# B&R Automation Studio project RS15_RX_30005_r00
Automation Studio 3.0.90.22 SP04; D.M. Le 24/08/2012 RS15_RX30005
Current program in the machine. End of commissioning. 
Customer IP config set

## Configuration Config1

CPU 5PPC2200.AL14-000, AutomationRuntime H4.91, Build 6.3.0, Safety 0.0, Vc V4.73.2

### Task classes (Cpu.sw)
```
Cyclic#1 (cycle 6000 us, tolerance 6000 us):
  GlobProgCa <- BagMachine_Section.GlobProgCalc.prg
  Alarms1 <- SupervisoryControl_Section.Alarm_Section.Alarms1.prg
  MainAlarms <- SupervisoryControl_Section.Alarm_Section.MainAlarms.prg
  Perf_Gen <- BagMachine_Section.Perf.Perf_Gen.prg
  A0_Basic <- BagMachine_Section.Servo_Power_Supply.Axis0.A0_Basic.prg
  A1_Basic <- BagMachine_Section.Perf.Axis1.A1_Basic.prg
  A2_Basic <- BagMachine_Section.FP.Axis2.A2_Basic.prg
  A3_Basic <- BagMachine_Section.Holding.Axis3.A3_Basic.prg
  A4_Basic <- BagMachine_Section.Tearing.Axis4.A4_Basic.prg
  A5_Basic <- BagMachine_Section.EntryPull.Axis5.A5_Basic.prg
  A5_Reg1 <- BagMachine_Section.EntryPull.Registration.A5_Reg1.prg
  A6_Basic <- BagMachine_Section.ExitPull.Axis6.A6_Basic.prg
  A7_Basic <- BagMachine_Section.Drum.Axis7.A7_Basic.prg
  A8_Basic <- BagMachine_Section.ColdMicroPerf.Axis8.A8_Basic.prg [disabled]
  A9_Basic <- BagMachine_Section.MasterAxis.A9_Init.A9_Basic.prg
  A11_Basic <- BagMachine_Section.Perf.Axis11_VirtualAxis.A11_Basic.prg
  A12_Basic <- BagMachine_Section.EnvBag.Axis12.A12_Basic.prg [disabled]
  A13_Basic <- BagMachine_Section.EnvBag.Axis13.A13_Basic.prg [disabled]
  A15_Basic <- BagMachine_Section.HotMicroPerf.Axis15.A15_Basic.prg [disabled]
  A1_Automat <- BagMachine_Section.Perf.Axis1.A1_Automat.prg
  A1_Automa1 <- BagMachine_Section.Perf.Axis1.A1_Automat2.prg
  A11_Automa <- BagMachine_Section.Perf.Axis11_VirtualAxis.A11_Automat.prg
  A2_Automat <- BagMachine_Section.FP.Axis2.A2_Automat.prg
  A3_Automat <- BagMachine_Section.Holding.Axis3.A3_Automat.prg
  A4_Automat <- BagMachine_Section.Tearing.Axis4.A4_Automat.prg
  A5_Automat <- BagMachine_Section.EntryPull.Axis5.A5_Automat.prg
  A6_Automat <- BagMachine_Section.ExitPull.Axis6.A6_Automat.prg
  A7_Automat <- BagMachine_Section.Drum.Axis7.A7_Automat.prg
  A8_Automat <- BagMachine_Section.ColdMicroPerf.Axis8.A8_Automat.prg [disabled]
  A12_Automa <- BagMachine_Section.EnvBag.Axis12.A12_Automat.prg [disabled]
  A13_Automa <- BagMachine_Section.EnvBag.Axis13.A13_Automat.prg [disabled]
  A15_Automa <- BagMachine_Section.HotMicroPerf.Axis15.A15_Automat.prg [disabled]
  Count <- BagMachine_Section.Count.prg
  SpeedLimit <- (binary)
Cyclic#2 (cycle 12000 us, tolerance 12000 us):
  A1_Control <- BagMachine_Section.Perf.Axis1.A1_Control.prg
  A1_Ref <- BagMachine_Section.Perf.Axis1.A1_Ref.prg
  A1_Cycle <- BagMachine_Section.Perf.Axis1.A1_Cycle.prg
  A11_Contro <- BagMachine_Section.Perf.Axis11_VirtualAxis.A11_Control.prg
  A2_Control <- BagMachine_Section.FP.Axis2.A2_Control.prg
  A2_Ref <- BagMachine_Section.FP.Axis2.A2_Ref.prg
  A2_Cycle <- BagMachine_Section.FP.Axis2.A2_Cycle.prg
  A3_Control <- BagMachine_Section.Holding.Axis3.A3_Control.prg
  A3_Ref <- BagMachine_Section.Holding.Axis3.A3_Ref.prg
  A3_Cycle <- BagMachine_Section.Holding.Axis3.A3_Cycle.prg
  A4_Control <- BagMachine_Section.Tearing.Axis4.A4_Control.prg
  A4_Ref <- BagMachine_Section.Tearing.Axis4.A4_Ref.prg
  A4_Cycle <- BagMachine_Section.Tearing.Axis4.A4_Cycle.prg
  A5_Control <- BagMachine_Section.EntryPull.Axis5.A5_Control.prg
  A5_Draw <- BagMachine_Section.EntryPull.Axis5.A5_Draw.prg
  A5_Reg2 <- BagMachine_Section.EntryPull.Registration.A5_Reg2.prg
  A6_Control <- BagMachine_Section.ExitPull.Axis6.A6_Control.prg
  A6_Draw <- BagMachine_Section.ExitPull.Axis6.A6_Draw.prg
  A7_Control <- BagMachine_Section.Drum.Axis7.A7_Control.prg
  A7_Ref <- BagMachine_Section.Drum.Axis7.A7_Ref.prg
  A7_Cycle <- BagMachine_Section.Drum.Axis7.A7_Cycle.prg
  A9_Control <- BagMachine_Section.MasterAxis.A9_Init.A9_Control.prg
  A8_Control <- BagMachine_Section.ColdMicroPerf.Axis8.A8_Control.prg [disabled]
  A8_Draw <- BagMachine_Section.ColdMicroPerf.Axis8.A8_Draw.prg [disabled]
  CMPerf_Gen <- BagMachine_Section.ColdMicroPerf.CMPerf_Gen.prg [disabled]
  A12_Contro <- BagMachine_Section.EnvBag.Axis12.A12_Control.prg [disabled]
  A12_Ref <- BagMachine_Section.EnvBag.Axis12.A12_Ref.prg [disabled]
  A12_Cycle <- BagMachine_Section.EnvBag.Axis12.A12_Cycle.prg [disabled]
  A13_Contro <- BagMachine_Section.EnvBag.Axis13.A13_Control.prg [disabled]
  A13_Ref <- BagMachine_Section.EnvBag.Axis13.A13_Ref.prg [disabled]
  A13_Cycle <- BagMachine_Section.EnvBag.Axis13.A13_Cycle.prg [disabled]
  A15_Contro <- BagMachine_Section.HotMicroPerf.Axis15.A15_Control.prg [disabled]
  A15_Ref <- BagMachine_Section.HotMicroPerf.Axis15.A15_Ref.prg [disabled]
  A15_Cycle <- BagMachine_Section.HotMicroPerf.Axis15.A15_Cycle.prg [disabled]
  A15_Motion <- BagMachine_Section.HotMicroPerf.Axis15.A15_MotionCycle.prg [disabled]
  HMPerf_Gen <- BagMachine_Section.HotMicroPerf.HMPerf_Gen.prg [disabled]
  Vacuum <- BagMachine_Section.Vacuum.prg
  Setup <- SupervisoryControl_Section.Setup.prg
  EntryNip <- BagMachine_Section.EntryPull.EntryNip.prg
  ExitNip <- BagMachine_Section.ExitPull.ExitNip.prg
  GlueTray <- BagMachine_Section.GlueTray.prg
  ColdGlue <- BagMachine_Section.ColdGlue.prg
  HotGlue <- BagMachine_Section.HotGlue.prg [disabled]
  RS_Glue <- BagMachine_Section.RS_Glue.prg [disabled]
  Unw_3W_Glu <- BagMachine_Section.Unw_3W_Glue.prg
  EB_Gen <- BagMachine_Section.EnvBag.EB_Gen.prg
  Guard_Mon <- SupervisoryControl_Section.Guard_Mon.prg
  Stop_Mon <- SupervisoryControl_Section.Stop_Mon.prg
  Servo_Mon <- SupervisoryControl_Section.Servo_Mon.prg
  EStopReset <- SupervisoryControl_Section.Alarm_Section.EStopReset.prg
  Jog <- SupervisoryControl_Section.Jog.prg
  Run <- SupervisoryControl_Section.Run.prg
  Warn_Horn <- SupervisoryControl_Section.Warn_Horn.prg
  Control <- BagMachine_Section.BagBundler.Control.prg
  Tilter <- BagMachine_Section.BagBundler.Tilter.prg
  Separator <- BagMachine_Section.BagBundler.Separator.prg
Cyclic#3 (cycle 20000 us, tolerance 20000 us):
  FP_Heater <- BagMachine_Section.FP.FP_Heater.prg
Cyclic#4:
  A1_CamProf <- BagMachine_Section.Perf.Axis1.A1_CamProfCalc.prg
  HMI_Contro <- HMI.HMI_Control.prg
  Units <- HMI.Units.prg
  Language <- HMI.Language.prg
  Splash <- HMI.Splash.prg
  Cmd_Trace <- HMI.Cmd_Trace.prg
  Recipe_1 <- HMI.Recipe_1.prg
  Recipe_2 <- HMI.Recipe_2.prg
  Message_1 <- HMI.Message_1.prg
  Message_2 <- HMI.Message_2.prg
  Password <- HMI.Password.prg
  PowerTimer <- SupervisoryControl_Section.PowerTimer.prg
  BackUp <- HMI.BackUp.prg
  Revision <- SupervisoryControl_Section.Revision.prg
  Speed <- SupervisoryControl_Section.Speed.prg
  CPURestart <- HMI.CPURestart.prg
  SetSpeedMo <- BagMachine_Section.MasterAxis.A9_Init.SetSpeedMode.prg
  ManMode <- SupervisoryControl_Section.ManMode.prg
  ExitTable <- BagMachine_Section.ExitTable.prg
  FP_Gen <- BagMachine_Section.FP.FP_Gen.prg
  Unwinder <- BagMachine_Section.Unwinder.prg
  3Web_Unit <- BagMachine_Section.3Web_Unit.prg
  FP_Dryer <- BagMachine_Section.FP.FP_Dryer.prg
Cyclic#7:
  HourMeter <- SupervisoryControl_Section.HourMeter.prg
DataObjects: arsdmsvg, arsdmhtm, arsdmsvp, Acp10sys
NcDataObjects: Error_Eng <- Error_Eng.dob, A0_Init <- BagMachine_Section.Servo_Power_Supply.Axis0.A0_Init.dob, A0_Par <- BagMachine_Section.Servo_Power_Supply.Axis0.A0_Par.dob, A1_Init <- BagMachine_Section.Perf.Axis1.A1_Init.dob, A1_Par <- BagMachine_Section.Perf.Axis1.A1_Par.dob, A2_Init <- BagMachine_Section.FP.Axis2.A2_Init.dob, A2_Par <- BagMachine_Section.FP.Axis2.A2_Par.dob, A3_Init <- BagMachine_Section.Holding.Axis3.A3_Init.dob, A3_Par <- BagMachine_Section.Holding.Axis3.A3_Par.dob, A4_Init <- BagMachine_Section.Tearing.Axis4.A4_Init.dob, A4_Par <- BagMachine_Section.Tearing.Axis4.A4_Par.dob, A5_Init <- BagMachine_Section.EntryPull.Axis5.A5_Init.dob, A5_Par <- BagMachine_Section.EntryPull.Axis5.A5_Par.dob, A6_Init <- BagMachine_Section.ExitPull.Axis6.A6_Init.dob, A6_Par <- BagMachine_Section.ExitPull.Axis6.A6_Par.dob, A7_Init <- BagMachine_Section.Drum.Axis7.A7_Init.dob, A7_Par <- BagMachine_Section.Drum.Axis7.A7_Par.dob, A8_Init <- BagMachine_Section.ColdMicroPerf.Axis8.A8_Init.dob [disabled], A8_Par <- BagMachine_Section.ColdMicroPerf.Axis8.A8_Par.dob [disabled], A9_Init <- BagMachine_Section.MasterAxis.A9_Init.A9_Init.dob, A9_Par <- BagMachine_Section.MasterAxis.A9_Init.A9_Par.dob, A11_Init <- BagMachine_Section.Perf.Axis11_VirtualAxis.A11_Init.dob, A11_Par <- BagMachine_Section.Perf.Axis11_VirtualAxis.A11_Par.dob, A12_Init <- BagMachine_Section.EnvBag.Axis12.A12_Init.dob [disabled], A12_Par <- BagMachine_Section.EnvBag.Axis12.A12_Par.dob [disabled], A13_Init <- BagMachine_Section.EnvBag.Axis13.A13_Init.dob [disabled], A13_Par <- BagMachine_Section.EnvBag.Axis13.A13_Par.dob [disabled], A15_Init <- BagMachine_Section.HotMicroPerf.Axis15.A15_Init.dob [disabled], A15_Par <- BagMachine_Section.HotMicroPerf.Axis15.A15_Par.dob [disabled], Axis1_Init, Axis1_par, Error_Engl, A0_Init1, A0_Par1
VcDataObjects: HMI_10 <- HMI.HMI_10.dob
Binaries: HMI_1002, HMI_1001, HMI_1003, vcbclass, vcpdpp30, vcpdsw, vcshared, vccdt, visvc, arialbi, vcresman, vcmgr, vcdsloc, vcptelo, webserv, arialbd, vcchspot, vccshape, vccpopup, vcdsint, vcalarm, vccddbox, vcnet, vcfntttf, vccbmp, vcclbox, vcctext, vcrt, vccbtn, vccstr, vcgclass, arial, vccline, vcpfmtcx, vcfile, vcpfpp30, vccovl, vccalarm, vctcal, vcpdvnc, vccnum, arsdm, iomap, sysconf, asfw, ashwd, arconfig, Acp10map, Acp10cfg, HMI_1502, HMI_1503, HMI_1501, vccpwd, HMI_601, HMI_602, HMI_603, vcvisapi, HMI_15, HMI_6, arialu_1, HMI_3, HMI_301, viscomp, ddpcxlk, aplib, HMI_302, vcinter
Libraries: Brsystem, AsMath, asstring, astime, FileIO, powerlnk, Visapi, HGWeber, Runtime, AsMem, CSV_File, AsIOAcc, AsARCfg, standard, sys_lib, convert, dataobj, Acp10man, Acp10par, NcGlobal, Acp10_MC, astcp, LoopConR
```

### Hardware
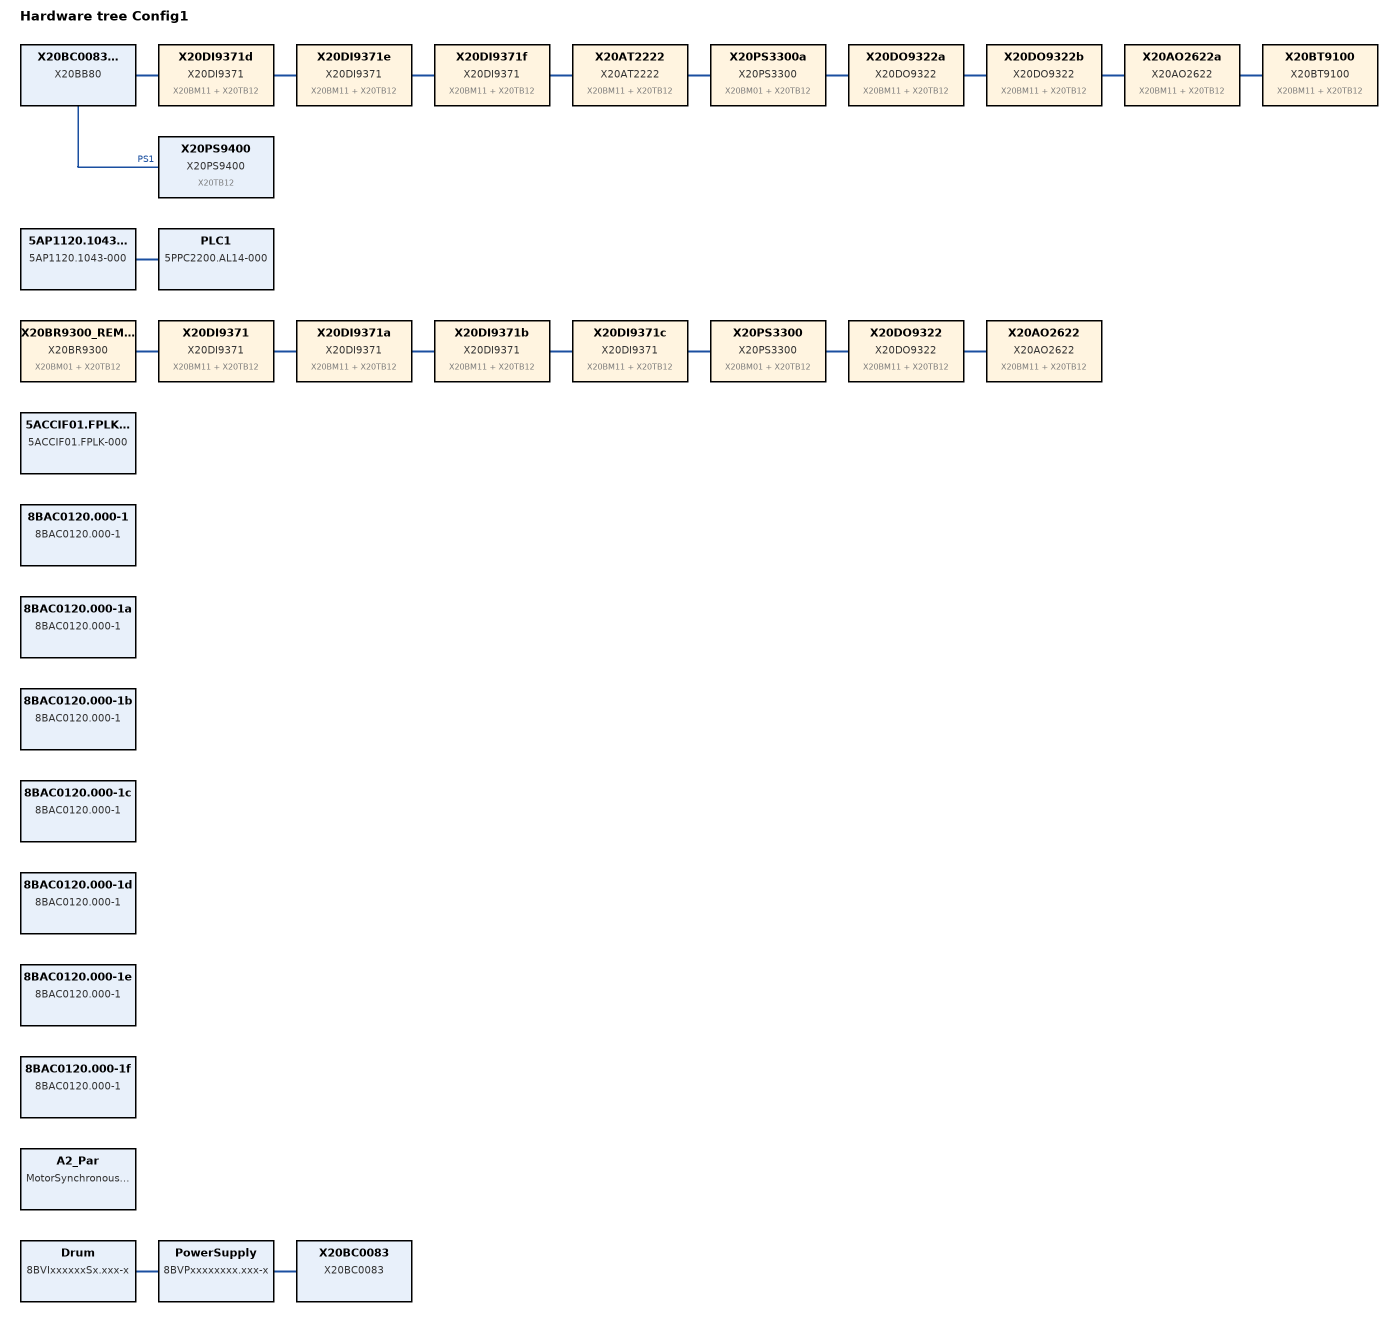
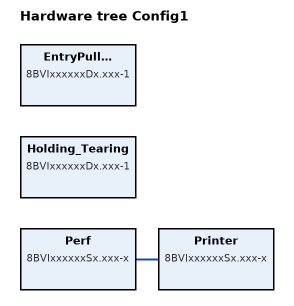
```
5ACCIF01.FPLK-000 : 5ACCIF01.FPLK-000 v1.9.0.0  [PLK2 -> X20BC0083.PLK2 [Cable Type=PowerlinkCable, Length=10, Version=1.0.0.3]; SL -> PLC1.SL1]
  Connector IF1:
    EplNatSubnet = 192.168.102.0
5AP1120.1043-000 : 5AP1120.1043-000 v2.1.0.0
  Connector IF20:
    AssignedOperatingSystem = ARemb
  Supervision = off
  VcObjectName = HMI_10
8BAC0120.000-1 : 8BAC0120.000-1 v2.2.0.0  [SS -> Perf.SS1]
8BAC0120.000-1a : 8BAC0120.000-1 v2.2.0.0  [SS -> Printer.SS1]
8BAC0120.000-1b : 8BAC0120.000-1 v2.2.0.0  [SS -> Holding_Tearing.SS1]
8BAC0120.000-1c : 8BAC0120.000-1 v2.2.0.0  [SS -> Holding_Tearing.SS2]
8BAC0120.000-1d : 8BAC0120.000-1 v2.2.0.0  [SS -> EntryPull_ExitPull.SS1]
8BAC0120.000-1e : 8BAC0120.000-1 v2.2.0.0  [SS -> EntryPull_ExitPull.SS2]
8BAC0120.000-1f : 8BAC0120.000-1 v2.2.0.0  [SS -> Drum.SS1]
A2_Par : MotorSynchronous_any v2.2.1.0 (Disabled=true)  [MT -> Printer.MT1]
  MOTOR_TYPE = 1
  MOTOR_COMPATIBILITY = 515
  MOTOR_POLEPAIRS = 2
  MOTOR_BRAKE_CURR_RATED = 0
  MOTOR_BRAKE_TORQ_RATED = 0
  MOTOR_BRAKE_ON_TIME = 0
  MOTOR_BRAKE_OFF_TIME = 0
  MOTOR_TEMPSENS_PAR1 = 391
  MOTOR_TEMPSENS_PAR2 = 1492
  MOTOR_TEMPSENS_PAR3 = -30
  MOTOR_TEMPSENS_PAR4 = 12.01
  MOTOR_TEMPSENS_PAR5 = 45.98
  MOTOR_TEMPSENS_PAR6 = 75.71
  MOTOR_TEMPSENS_PAR7 = 102.2
  MOTOR_TEMPSENS_PAR8 = 126.41
  MOTOR_TEMPSENS_PAR9 = 148.88
  MOTOR_TEMPSENS_PAR10 = 170
  MOTOR_VOLTAGE_RATED = 322
  MOTOR_VOLTAGE_CONST = 0
  MOTOR_SPEED_RATED = 1000
  MOTOR_SPEED_MAX = 8000
  MOTOR_TORQ_STALL = 162,34
  MOTOR_TORQ_RATED = 162.34
  MOTOR_TORQ_MAX = 577.34
  MOTOR_TORQ_CONST = 0
  MOTOR_CURR_STALL = 40.69
  MOTOR_CURR_RATED = 40.69
  MOTOR_CURR_MAX = 238.47
  MOTOR_WIND_CROSS_SECT = 0
  MOTOR_STATOR_RESISTANCE = 0.1542
  MOTOR_STATOR_INDUCTANCE = 0.00180
  MOTOR_INERTIA = 0
  MOTOR_COMMUT_OFFSET = 0
  MOTOR_TAU_THERM = 0
  MOTOR_WIND_TEMP_MAX = 100
Drum : 8BVIxxxxxxSx.xxx-x v2.3.0.0  [PLK1 -> EntryPull_ExitPull.PLK2 (NodeNumber=7) [Cable Type=PowerlinkCable, Length=10, Version=1.0.0.3]; PLK2 -> PowerSupply.PLK1 (NodeNumber=7) [Cable Type=PowerlinkCable, Length=10, Version=1.0.0.3]]
  SupplyVoltage = 565
EntryPull_ExitPull : 8BVIxxxxxxDx.xxx-1 v2.3.0.2  [PLK1 -> Holding_Tearing.PLK2 (NodeNumber=5) [Cable Type=PowerlinkCable, Length=10, Version=1.0.0.3]; PLK2 -> Drum.PLK1 (NodeNumber=5) [Cable Type=PowerlinkCable, Length=10, Version=1.0.0.3]]
Holding_Tearing : 8BVIxxxxxxDx.xxx-1 v2.3.0.2  [PLK1 -> Printer.PLK2 (NodeNumber=3) [Cable Type=PowerlinkCable, Length=10, Version=1.0.0.3]; PLK2 -> EntryPull_ExitPull.PLK1 (NodeNumber=3) [Cable Type=PowerlinkCable, Length=10, Version=1.0.0.3]]
PLC1 : 5PPC2200.AL14-000 v2.0.7.0  [SY -> 5AP1120.1043-000.SY1]
  Connector IF3:
    AssignedOperatingSystem = ARemb
    ActivateDevice = 1
    Mode = Manual
    InternetAddress = 10.0.1.67
    SubnetMask = 255.255.255.0
    Vnc1
    VncVcObjectName1 = HMI_10
    VncAuthentication1 = 1
    VncPasswordViewOnly1 = 725
    VncPasswordViewControl1 = 4444
    VncMaxConnections1 = 4
    VncRefreshRate1 = 200
    VncConnectionTimeout1 = 20
  Connector IF4:
    AssignedOperatingSystem = ARemb
    ActivateDevice = 1
  Connector IF5:
    AssignedOperatingSystem = ARemb
  Connector IF6:
    AssignedOperatingSystem = ARemb
  ConfigurationID = RS15_RX_30005_r00_Config1
  UserPartitionSize = 0
  UserRamDevice = PCI.1.PPC21xx.SRAM
  UserRamSize = 477648
  RemMemDevice = PCI.1.PPC21xx.SRAM
  RemMemSize = 30000
  PermanentPvSize = 1548
  RemanentGlobalPvSize = 20000
  VolatileGlobalPvSize = 25000
  TimerDeviceType = EPLX2X
  TimerDevice = 5ACCIF01.FPLK-000.IF1
  IdleTaskClass = 8
  TaskClassIdleTime = 4000
  XLinkUseDefault = 0
  XLinkDuration = 2000
  Cyclic1Duration = 6000
  Cyclic1Tolerance = 6000
  Cyclic2Duration = 12000
  Cyclic2Tolerance = 12000
  Cyclic3Duration = 20000
  Cyclic3Tolerance = 20000
  FileDevice1
  FileDeviceName1 = USB1
  FileDevicePath1 = IF6.ST1
  FileDevice2
  FileDeviceName2 = USB2
  FileDevicePath2 = IF7.ST1
  TimeZone = 50
  EthernetHostName = RS15-30005
  EthernetDefaultGateway = 10.0.1.1
  ActivateDns = 1
  DnsDefaultDomain = x
  DnsServer1 = 10.0.1.15
  FtpUser1
  FtpUsername1 = weber
  FtpUserPassword1 = uro1CudS6bYO7XlsqDVBWd16H3OnXC5QTtArHRz3m8w=  // tech725
  FtpUserSalt1 = 2plUcaTe
Perf : 8BVIxxxxxxSx.xxx-x v2.3.0.0  [PLK2 -> Printer.PLK1 (NodeNumber=1) [Cable Type=PowerlinkCable, Length=10, Version=1.0.0.3]]
  SupplyVoltage = 565
PowerSupply : 8BVPxxxxxxxx.xxx-x v2.3.0.0  [PLK1 -> Drum.PLK2 (NodeNumber=10) [Cable Type=PowerlinkCable, Length=10, Version=1.0.0.3]; PLK2 -> X20BC0083.PLK1 (NodeNumber=10) [Cable Type=PowerlinkCable, Length=10, Version=1.0.0.3]]
Printer : 8BVIxxxxxxSx.xxx-x v2.3.0.0  [PLK1 -> Perf.PLK2 (NodeNumber=2) [Cable Type=PowerlinkCable, Length=10, Version=1.0.0.3]; PLK2 -> Holding_Tearing.PLK1 (NodeNumber=2) [Cable Type=PowerlinkCable, Length=10, Version=1.0.0.3]]
  SupplyVoltage = 565
X20AO2622 : X20AO2622 v1.4.1.0  [SS1 -> X20TB12o.SS; SL -> X20BM11l.SL1]
  FunctionModel = Standard
  Supervision = off
X20AO2622a : X20AO2622 v1.4.1.0  [SS1 -> X20TB12g.SS; SL -> X20BM11f.SL1]
  FunctionModel = Standard
  Supervision = off
X20AT2222 : X20AT2222 v1.6.0.0  [SS1 -> X20TB12c.SS; SL -> X20BM11c.SL1]
  FunctionModel = FunctionModel001
  Supervision = off
X20BC0083 : X20BC0083 v2.11.1.0  [PLK1 -> PowerSupply.PLK2 (NodeNumber=11) [Cable Type=PowerlinkCable, Length=10, Version=1.0.0.3]; PLK2 -> 5ACCIF01.FPLK-000.PLK2 (NodeNumber=11) [Cable Type=PowerlinkCable, Length=10, Version=1.0.0.3]; SL -> X20BC0083_MainEnclosureREM_IO_E1.SL1]
  Supervision = off
  Multiplexed = 1
X20BC0083_MainEnclosureREM_IO_E1 : X20BB80 v1.1.0.0
X20BM01 : X20BM01 v2.2.0.0  [X2X1 -> X20BM11c.X2X2]
X20BM01a : X20BM01 v2.2.0.0
X20BM01b : X20BM01 v2.2.0.0  [X2X1 -> X20BM11j.X2X2]
X20BM11 : X20BM11 v1.0.0.1  [X2X1 -> X20BC0083_MainEnclosureREM_IO_E1.IF1]
X20BM11a : X20BM11 v1.0.0.1  [X2X1 -> X20BM11.X2X2]
X20BM11b : X20BM11 v1.0.0.1  [X2X1 -> X20BM11a.X2X2]
X20BM11c : X20BM11 v1.0.0.1  [X2X1 -> X20BM11b.X2X2]
X20BM11d : X20BM11 v1.0.0.1  [X2X1 -> X20BM01.X2X2]
X20BM11e : X20BM11 v1.0.0.1  [X2X1 -> X20BM11d.X2X2]
X20BM11f : X20BM11 v1.0.0.1  [X2X1 -> X20BM11e.X2X2]
X20BM11g : X20BM11 v1.0.0.1  [X2X1 -> X20BM01a.X2X2]
X20BM11h : X20BM11 v1.0.0.1  [X2X1 -> X20BM11g.X2X2]
X20BM11i : X20BM11 v1.0.0.1  [X2X1 -> X20BM11h.X2X2]
X20BM11j : X20BM11 v1.0.0.1  [X2X1 -> X20BM11i.X2X2]
X20BM11k : X20BM11 v1.0.0.1  [X2X1 -> X20BM01b.X2X2]
X20BM11l : X20BM11 v1.0.0.1  [X2X1 -> X20BM11k.X2X2]
X20BM11m : X20BM11 v1.0.0.1  [X2X1 -> X20BM11f.X2X2]
X20BR9300_REM_IO_L3 : X20BR9300 v1.0.3.0  [SS1 -> X20TB12p.SS; SL -> X20BM01a.SL1; X2X1 -> X20BT9100.X2X1 [Cable Type=X2XCable, Length=10, Version=1.0.0.3]]
  Supervision = off
X20BT9100 : X20BT9100 v1.3.0.0  [SS1 -> X20TB12q.SS; SL -> X20BM11m.SL1]
  Supervision = off
X20DI9371 : X20DI9371 v1.6.0.0  [SS1 -> X20TB12i.SS; SL -> X20BM11g.SL1]
  Supervision = off
X20DI9371a : X20DI9371 v1.6.0.0  [SS1 -> X20TB12j.SS; SL -> X20BM11h.SL1]
  Supervision = off
X20DI9371b : X20DI9371 v1.6.0.0  [SS1 -> X20TB12k.SS; SL -> X20BM11i.SL1]
  Supervision = off
X20DI9371c : X20DI9371 v1.6.0.0  [SS1 -> X20TB12l.SS; SL -> X20BM11j.SL1]
  Supervision = off
X20DI9371d : X20DI9371 v1.6.0.0  [SS1 -> X20TB12.SS; SL -> X20BM11.SL1]
  Supervision = off
X20DI9371e : X20DI9371 v1.6.0.0  [SS1 -> X20TB12a.SS; SL -> X20BM11a.SL1]
  Supervision = off
X20DI9371f : X20DI9371 v1.6.0.0  [SS1 -> X20TB12b.SS; SL -> X20BM11b.SL1]
  Supervision = off
X20DO9322 : X20DO9322 v1.6.0.0  [SS1 -> X20TB12n.SS; SL -> X20BM11k.SL1]
  Supervision = off
X20DO9322a : X20DO9322 v1.6.0.0  [SS1 -> X20TB12e.SS; SL -> X20BM11d.SL1]
  Supervision = off
X20DO9322b : X20DO9322 v1.6.0.0  [SS1 -> X20TB12f.SS; SL -> X20BM11e.SL1]
  Supervision = off
X20PS3300 : X20PS3300 v1.2.0.0  [SS1 -> X20TB12m.SS; SL -> X20BM01b.SL1]
  Supervision = off
X20PS3300a : X20PS3300 v1.2.0.0  [SS1 -> X20TB12d.SS; SL -> X20BM01.SL1]
  Supervision = off
X20PS9400 : X20PS9400 v1.8.0.0  [SS1 -> X20TB12h.SS; PS -> X20BC0083_MainEnclosureREM_IO_E1.PS1]
  Supervision = off
X20TB12 : X20TB12 v1.0.0.0
X20TB12a : X20TB12 v1.0.0.0
X20TB12b : X20TB12 v1.0.0.0
X20TB12c : X20TB12 v1.0.0.0
X20TB12d : X20TB12 v1.0.0.0
X20TB12e : X20TB12 v1.0.0.0
X20TB12f : X20TB12 v1.0.0.0
X20TB12g : X20TB12 v1.0.0.0
X20TB12h : X20TB12 v1.0.0.0
X20TB12i : X20TB12 v1.0.0.0
X20TB12j : X20TB12 v1.0.0.0
X20TB12k : X20TB12 v1.0.0.0
X20TB12l : X20TB12 v1.0.0.0
X20TB12m : X20TB12 v1.0.0.0
X20TB12n : X20TB12 v1.0.0.0
X20TB12o : X20TB12 v1.0.0.0
X20TB12p : X20TB12 v1.0.0.0
X20TB12q : X20TB12 v1.0.0.0
```

### Cpu.per - PLC1/Cpu.per
```iecst
(********************************************************************
 * COPYRIGHT --
 ********************************************************************
 * File: Cpu.per
 * Author: pkiel
 * Created: September 02, 2009
 ********************************************************************
 * Declaration of permanent variables
 ********************************************************************)
VAR_CONFIG
	gEndPosData AT %M0;
	gMachineTime AT %M720;
  gSP_A AT %M832;
END_VAR
```

### IoMap.iom - PLC1/IoMap.iom
```iecst
(********************************************************************
 * COPYRIGHT --
 ********************************************************************
 * File: IoMap.iom
 * Author: pkiel
 * Created: September 02, 2009
 ********************************************************************
 * IO mapping file
 ********************************************************************)
VAR_CONFIG
	Alarms1.stModuleOK_IO_E1_Slot[1].bStat AT %IX.SL1.SS1.IF2.ST11.ModuleOk;
	Alarms1.stModuleOK_IO_E1_Slot[2].bStat AT %IX.SL1.SS1.IF2.ST11.IF1.ST1.ModuleOk;
	Alarms1.stModuleOK_IO_L3_Slot[1].bStat AT %IX.SL1.SS1.IF1.ST1.ModuleOk;
	Alarms1.stModuleOK_IO_E1_Slot[7].bStat AT %IX.SL1.SS1.IF2.ST11.IF1.ST6.ModuleOk;
	Alarms1.stModuleOK_IO_E1_Slot[10].bStat AT %IX.SL1.SS1.IF2.ST11.IF1.ST9.ModuleOk;
	gQ_CMD_RS_ExitTableSpeed AT %QW.SL1.SS1.IF2.ST11.IF1.ST9.AnalogOutput02;
	gQ_CMD_UNW_GluePressure AT %QW.SL1.SS1.IF2.ST11.IF1.ST9.AnalogOutput01;
	gI_StopPB_2 AT %IX.SL1.SS1.IF1.ST2.DigitalInput01;
	Alarms1.stModuleOK_IO_L3_Slot[2].bStat AT %IX.SL1.SS1.IF1.ST2.ModuleOk;
	gI_EstopPB_1 AT %IX.SL1.SS1.IF1.ST2.DigitalInput02;
	gI_SS_PerfPos AT %IX.SL1.SS1.IF1.ST2.DigitalInput04;
	gI_SS_PerfNeg AT %IX.SL1.SS1.IF1.ST2.DigitalInput03;
	gI_PB_MachineStart AT %IX.SL1.SS1.IF1.ST2.DigitalInput05;
	gI_FasterPB_1 AT %IX.SL1.SS1.IF1.ST2.DigitalInput06;
	gI_SS_GluePanUpDown AT %IX.SL1.SS1.IF1.ST2.DigitalInput07;
	gI_SS_WebExitNip AT %IX.SL1.SS1.IF1.ST2.DigitalInput08;
	gI_PrintOff_PB AT %IX.SL1.SS1.IF1.ST2.DigitalInput09;
	gI_PrintOn_PB AT %IX.SL1.SS1.IF1.ST2.DigitalInput10;
	gI_SS_TearingNeg AT %IX.SL1.SS1.IF1.ST2.DigitalInput11;
	gI_SS_TearingPos AT %IX.SL1.SS1.IF1.ST2.DigitalInput12;
	Alarms1.stModuleOK_IO_L3_Slot[3].bStat AT %IX.SL1.SS1.IF1.ST3.ModuleOk;
	gI_SS_HoldingNeg AT %IX.SL1.SS1.IF1.ST3.DigitalInput01;
	gI_SS_HoldingPos AT %IX.SL1.SS1.IF1.ST3.DigitalInput02;
	gI_SS_ExitTableSlower AT %IX.SL1.SS1.IF1.ST3.DigitalInput03;
	gI_SS_ExitTableFaster AT %IX.SL1.SS1.IF1.ST3.DigitalInput04;
	gI_EstopPB_2 AT %IX.SL1.SS1.IF1.ST3.DigitalInput05;
	gI_SlowerPB_2 AT %IX.SL1.SS1.IF1.ST3.DigitalInput06;
	gI_JamPE_RS AT %IX.SL1.SS1.IF1.ST3.DigitalInput07;
	gI_GSW_Door1 AT %IX.SL1.SS1.IF1.ST3.DigitalInput09;
	gI_JogPB_1 AT %IX.SL1.SS1.IF1.ST3.DigitalInput08;
	gI_GSW_Door2 AT %IX.SL1.SS1.IF1.ST3.DigitalInput10;
	gI_GSW_Tearing AT %IX.SL1.SS1.IF1.ST3.DigitalInput11;
	gI_GSW_Drum AT %IX.SL1.SS1.IF1.ST3.DigitalInput12;
	Alarms1.stModuleOK_IO_L3_Slot[4].bStat AT %IX.SL1.SS1.IF1.ST4.ModuleOk;
	gI_FstopPB_1 AT %IX.SL1.SS1.IF1.ST4.DigitalInput01;
	gI_SS_DrumPos AT %IX.SL1.SS1.IF1.ST4.DigitalInput02;
	gI_SS_DrumNeg AT %IX.SL1.SS1.IF1.ST4.DigitalInput03;
	gI_SS_SeamGlueOnOff AT %IX.SL1.SS1.IF1.ST4.DigitalInput04;
	gI_SS_WebEntryNipOn_1 AT %IX.SL1.SS1.IF1.ST4.DigitalInput05;
	gI_SS_WebEntryNipOff_1 AT %IX.SL1.SS1.IF1.ST4.DigitalInput06;
	gI_SS_WebEntryNipOn_2 AT %IX.SL1.SS1.IF1.ST4.DigitalInput07;
	gI_SS_WebEntryNipOff_2 AT %IX.SL1.SS1.IF1.ST4.DigitalInput08;
	gI_ResetPB_1 AT %IX.SL1.SS1.IF1.ST4.DigitalInput09;
	gI_EstopPB_3 AT %IX.SL1.SS1.IF1.ST4.DigitalInput10;
	gI_AirPressureOK AT %IX.SL1.SS1.IF1.ST4.DigitalInput11;
	gI_WebBreakPE_1 AT %IX.SL1.SS1.IF1.ST4.DigitalInput12;
	Alarms1.stModuleOK_IO_L3_Slot[9].bStat AT %IX.SL1.SS1.IF1.ST8.ModuleOk;
	Alarms1.stModuleOK_IO_L3_Slot[8].bStat AT %IX.SL1.SS1.IF1.ST8.ModuleOk;
	Alarms1.stModuleOK_IO_L3_Slot[7].bStat AT %IX.SL1.SS1.IF1.ST7.ModuleOk;
	gQ_SOL_BagCount AT %QX.SL1.SS1.IF1.ST7.DigitalOutput01;
	gQ_SOL_WebExitNip AT %QX.SL1.SS1.IF1.ST7.DigitalOutput02;
	gQ_SOL_GluePan AT %QX.SL1.SS1.IF1.ST7.DigitalOutput03;
	gQ_L3_Spare1 AT %QX.SL1.SS1.IF1.ST7.DigitalOutput04;
	gQ_SOL_WebEntryNip AT %QX.SL1.SS1.IF1.ST7.DigitalOutput05;
	gQ_PL_MainPower AT %QX.SL1.SS1.IF1.ST7.DigitalOutput06;
	gQ_PL_GenFailure AT %QX.SL1.SS1.IF1.ST7.DigitalOutput07;
	gQ_L3_Spare2 AT %QX.SL1.SS1.IF1.ST7.DigitalOutput08;
	gQ_L3_Spare3 AT %QX.SL1.SS1.IF1.ST7.DigitalOutput09;
	gQ_L3_Spare4 AT %QX.SL1.SS1.IF1.ST7.DigitalOutput10;
	gQ_L3_Spare5 AT %QX.SL1.SS1.IF1.ST7.DigitalOutput11;
	gQ_L3_Spare6 AT %QX.SL1.SS1.IF1.ST7.DigitalOutput12;
	Alarms1.stModuleOK_IO_L3_Slot[6].bStat AT %IX.SL1.SS1.IF1.ST6.ModuleOk;
	Alarms1.stModuleOK_IO_L3_Slot[5].bStat AT %IX.SL1.SS1.IF1.ST5.ModuleOk;
	gI_SS_MainPowerOn AT %IX.SL1.SS1.IF1.ST5.DigitalInput01;
	gI_SS_MainPowerOff AT %IX.SL1.SS1.IF1.ST5.DigitalInput02;
	gI_EstopPB_4 AT %IX.SL1.SS1.IF1.ST5.DigitalInput03;
	gI_EstopPB_5 AT %IX.SL1.SS1.IF1.ST5.DigitalInput04;
	gI_GSW_PerfDoors AT %IX.SL1.SS1.IF1.ST5.DigitalInput05;
	gI_GSW_RSEntry AT %IX.SL1.SS1.IF1.ST5.DigitalInput07;
	gI_StopPB_3 AT %IX.SL1.SS1.IF1.ST5.DigitalInput09;
	gI_JogPB_2 AT %IX.SL1.SS1.IF1.ST5.DigitalInput10;
	gI_L3_Spare1 AT %IX.SL1.SS1.IF1.ST5.DigitalInput06;
	gI_L3_Spare2 AT %IX.SL1.SS1.IF1.ST5.DigitalInput08;
	gI_L3_Spare3 AT %IX.SL1.SS1.IF1.ST5.DigitalInput11;
	gI_L3_Spare4 AT %IX.SL1.SS1.IF1.ST5.DigitalInput12;
	gQ_CMD_RS_GluePressure AT %QW.SL1.SS1.IF1.ST8.AnalogOutput01;
	gAQ_L3_Spare1 AT %QW.SL1.SS1.IF1.ST8.AnalogOutput02;
	Alarms1.stModuleOK_IO_E1_Slot[3].bStat AT %IX.SL1.SS1.IF2.ST11.IF1.ST2.ModuleOk;
	Alarms1.stModuleOK_IO_E1_Slot[4].bStat AT %IX.SL1.SS1.IF2.ST11.IF1.ST3.ModuleOk;
	Alarms1.stModuleOK_IO_E1_Slot[5].bStat AT %IX.SL1.SS1.IF2.ST11.IF1.ST4.ModuleOk;
	Alarms1.stModuleOK_IO_E1_Slot[6].bStat AT %IX.SL1.SS1.IF2.ST11.IF1.ST5.ModuleOk;
	Alarms1.stModuleOK_IO_E1_Slot[8].bStat AT %IX.SL1.SS1.IF2.ST11.IF1.ST7.ModuleOk;
	Alarms1.stModuleOK_IO_E1_Slot[9].bStat AT %IX.SL1.SS1.IF2.ST11.IF1.ST8.ModuleOk;
	gI_SafetyRelay_EStopOK AT %IX.SL1.SS1.IF2.ST11.IF1.ST2.DigitalInput01;
	gI_JogPB_3 AT %IX.SL1.SS1.IF2.ST11.IF1.ST2.DigitalInput02;
	gI_StopPB_1 AT %IX.SL1.SS1.IF2.ST11.IF1.ST2.DigitalInput03;
	gI_SafetyRelay_GuardOK AT %IX.SL1.SS1.IF2.ST11.IF1.ST2.DigitalInput04;
	gI_SlowerPB_1 AT %IX.SL1.SS1.IF2.ST11.IF1.ST2.DigitalInput05;
	gI_E1_Spare1 AT %IX.SL1.SS1.IF2.ST11.IF1.ST2.DigitalInput06;
	gI_E1_Spare2 AT %IX.SL1.SS1.IF2.ST11.IF1.ST2.DigitalInput07;
	gI_230Vac_OK AT %IX.SL1.SS1.IF2.ST11.IF1.ST2.DigitalInput08;
	gI_E1_Spare3 AT %IX.SL1.SS1.IF2.ST11.IF1.ST2.DigitalInput12;
	gI_MP_GlueSlowRotation AT %IX.SL1.SS1.IF2.ST11.IF1.ST2.DigitalInput09;
	gI_MP_Vacuum AT %IX.SL1.SS1.IF2.ST11.IF1.ST2.DigitalInput10;
	gI_MP_PerfFan AT %IX.SL1.SS1.IF2.ST11.IF1.ST2.DigitalInput11;
	gI_SS_FP_NipRol AT %IX.SL1.SS1.IF2.ST11.IF1.ST3.DigitalInput01;
	gI_MP_FP_MotorFan AT %IX.SL1.SS1.IF2.ST11.IF1.ST3.DigitalInput02;
	gI_FP_PrintOn_PB AT %IX.SL1.SS1.IF2.ST11.IF1.ST3.DigitalInput03;
	gI_FP_PrintOff_PB AT %IX.SL1.SS1.IF2.ST11.IF1.ST3.DigitalInput04;
	gI_MP_FP_SlowRot1 AT %IX.SL1.SS1.IF2.ST11.IF1.ST3.DigitalInput05;
	gI_MP_FP_SlowRot2 AT %IX.SL1.SS1.IF2.ST11.IF1.ST3.DigitalInput06;
	gI_MP_FP_SlowRot3 AT %IX.SL1.SS1.IF2.ST11.IF1.ST3.DigitalInput07;
	gI_MP_FP_SlowRot4 AT %IX.SL1.SS1.IF2.ST11.IF1.ST3.DigitalInput08;
	gI_GSW_FP_Doors AT %IX.SL1.SS1.IF2.ST11.IF1.ST3.DigitalInput09;
	gI_GSW_FP_Gates AT %IX.SL1.SS1.IF2.ST11.IF1.ST3.DigitalInput10;
	gI_E1_Spare4 AT %IX.SL1.SS1.IF2.ST11.IF1.ST3.DigitalInput11;
	gI_E1_Spare5 AT %IX.SL1.SS1.IF2.ST11.IF1.ST3.DigitalInput12;
	gI_EstopPB_Unwind AT %IX.SL1.SS1.IF2.ST11.IF1.ST4.DigitalInput04;
	gI_E1_Spare6 AT %IX.SL1.SS1.IF2.ST11.IF1.ST4.DigitalInput03;
	gI_E1_Spare7 AT %IX.SL1.SS1.IF2.ST11.IF1.ST4.DigitalInput05;
	gI_E1_Spare8 AT %IX.SL1.SS1.IF2.ST11.IF1.ST4.DigitalInput09;
	gI_SS_UNW_ForkUp AT %IX.SL1.SS1.IF2.ST11.IF1.ST4.DigitalInput01;
	gI_SS_UNW_ForkDown AT %IX.SL1.SS1.IF2.ST11.IF1.ST4.DigitalInput02;
	gI_UNW_EndReelPapPE AT %IX.SL1.SS1.IF2.ST11.IF1.ST4.DigitalInput06;
	gI_SS_UNW_Brake AT %IX.SL1.SS1.IF2.ST11.IF1.ST4.DigitalInput07;
	gI_MP_UNW_HydroPump AT %IX.SL1.SS1.IF2.ST11.IF1.ST4.DigitalInput08;
	gI_MP_DRY_Blower AT %IX.SL1.SS1.IF2.ST11.IF1.ST4.DigitalInput12;
	gI_MP_DRY_Heater AT %IX.SL1.SS1.IF2.ST11.IF1.ST4.DigitalInput11;
	gI_DRY_Thermostat AT %IX.SL1.SS1.IF2.ST11.IF1.ST4.DigitalInput10;
	gAI_DRY_Pt100_Temp AT %IW.SL1.SS1.IF2.ST11.IF1.ST5.Temperature01;
	gAI_E1_Spare1 AT %IW.SL1.SS1.IF2.ST11.IF1.ST5.Temperature02;
	gQ_CR_WarningHorn AT %QX.SL1.SS1.IF2.ST11.IF1.ST7.DigitalOutput01;
	gQ_CR_EstopReset AT %QX.SL1.SS1.IF2.ST11.IF1.ST7.DigitalOutput02;
	gQ_CR_WatchDog AT %QX.SL1.SS1.IF2.ST11.IF1.ST7.DigitalOutput03;
	gQ_CR_MainPowerOn AT %QX.SL1.SS1.IF2.ST11.IF1.ST7.DigitalOutput04;
	gQ_CON_Vacuum AT %QX.SL1.SS1.IF2.ST11.IF1.ST7.DigitalOutput05;
	gQ_CON_GlueSlowRotation AT %QX.SL1.SS1.IF2.ST11.IF1.ST7.DigitalOutput06;
	gQ_CR_GuardBypass AT %QX.SL1.SS1.IF2.ST11.IF1.ST7.DigitalOutput07;
	gQ_E1_Spare1 AT %QX.SL1.SS1.IF2.ST11.IF1.ST7.DigitalOutput08;
	gQ_E1_Spare2 AT %QX.SL1.SS1.IF2.ST11.IF1.ST7.DigitalOutput10;
	gQ_E1_Spare3 AT %QX.SL1.SS1.IF2.ST11.IF1.ST7.DigitalOutput11;
	gQ_E1_Spare4 AT %QX.SL1.SS1.IF2.ST11.IF1.ST7.DigitalOutput12;
	gQ_CR_ColdGlue AT %QX.SL1.SS1.IF2.ST11.IF1.ST7.DigitalOutput09;
	gQ_CR_FP_Print AT %QX.SL1.SS1.IF2.ST11.IF1.ST8.DigitalOutput02;
	gQ_CR_FP_NipRol AT %QX.SL1.SS1.IF2.ST11.IF1.ST8.DigitalOutput01;
	gQ_CR_UNW_HydroPump AT %QX.SL1.SS1.IF2.ST11.IF1.ST8.DigitalOutput03;
	gQ_CR_UNW_PIDRegul AT %QX.SL1.SS1.IF2.ST11.IF1.ST8.DigitalOutput04;
	gQ_CR_UNW_Brake AT %QX.SL1.SS1.IF2.ST11.IF1.ST8.DigitalOutput05;
	gI_SS_UNW_ForkUp AT %QX.SL1.SS1.IF2.ST11.IF1.ST8.DigitalOutput06;
	gI_SS_UNW_ForkDown AT %QX.SL1.SS1.IF2.ST11.IF1.ST8.DigitalOutput07;
	gQ_CR_DRY_Blower AT %QX.SL1.SS1.IF2.ST11.IF1.ST8.DigitalOutput10;
	gQ_CR_DRY_HeatContinu AT %QX.SL1.SS1.IF2.ST11.IF1.ST8.DigitalOutput09;
	gQ_CR_DRY_HeatRegul AT %QX.SL1.SS1.IF2.ST11.IF1.ST8.DigitalOutput08;
	gQ_E1_Spare5 AT %QX.SL1.SS1.IF2.ST11.IF1.ST8.DigitalOutput11;
	gQ_E1_Spare6 AT %QX.SL1.SS1.IF2.ST11.IF1.ST8.DigitalOutput12;
	g_usiAI_DRY_Pt100_TempStatus AT %IB.SL1.SS1.IF2.ST11.IF1.ST5.StatusInput01;
END_VAR
```

### Acp10cfg.ncc - PLC1/Motion/Acp10cfg.ncc
```
NcConfiguration (Version=2.14.0, NcSwId=acp10)
  ACP10CF1_typ:
    cnt_nettrc_rec_drive = 500
    bufsize_trace_upload = 1200
    tc_nc_man_task = Cyclic #1
    glob_pv_as_ncobject = Yes
    network_init:
      ncsw_init_execute = Yes
      automatic_execute = No
      node_nr_warning = Yes
      net_err_before_ncact = Yes
    nettrc:
      enter_parsecrec = Yes
      enter_ncaction = Yes
      save_ring_startidx = No
    plk_if[0]:
      if_name = SL1.SS1.IF2
```

### Acp10map.ncm - PLC1/Motion/Acp10map.ncm
```
NcMapping (NcSwId=acp10)
  NcObject Axis3 (ModuleAddress=SL1.SS1.IF2.ST3, InterfaceType=Powerlink, Type=ncAXIS, Channel=1, InitParameter=A3_Init, AcoposParameter=A3_Par, Disabled=FALSE, ModuleDisabled=FALSE)
  NcObject SL1.SS1.IF2.ST3.VAxis1 (ModuleAddress=SL1.SS1.IF2.ST3, InterfaceType=Powerlink, Type=ncV_AXIS, Channel=1, Disabled=TRUE, ModuleDisabled=FALSE)
  NcObject Axis4 (ModuleAddress=SL1.SS1.IF2.ST3, InterfaceType=Powerlink, Type=ncAXIS, Channel=2, InitParameter=A4_Init, AcoposParameter=A4_Par, Disabled=FALSE, ModuleDisabled=FALSE)
  NcObject SL1.SS1.IF2.ST3.VAxis2 (ModuleAddress=SL1.SS1.IF2.ST3, InterfaceType=Powerlink, Type=ncV_AXIS, Channel=2, Disabled=TRUE, ModuleDisabled=FALSE)
  NcObject Axis5 (ModuleAddress=SL1.SS1.IF2.ST5, InterfaceType=Powerlink, Type=ncAXIS, Channel=1, InitParameter=A5_Init, AcoposParameter=A5_Par, Disabled=FALSE, ModuleDisabled=FALSE)
  NcObject Axis9 (ModuleAddress=SL1.SS1.IF2.ST5, InterfaceType=Powerlink, Type=ncV_AXIS, Channel=1, InitParameter=A9_Init, AcoposParameter=A9_Par, Disabled=FALSE, ModuleDisabled=FALSE)
  NcObject Axis6 (ModuleAddress=SL1.SS1.IF2.ST5, InterfaceType=Powerlink, Type=ncAXIS, Channel=2, InitParameter=A6_Init, AcoposParameter=A6_Par, Disabled=FALSE, ModuleDisabled=FALSE)
  NcObject SL1.SS1.IF2.ST5.VAxis2 (ModuleAddress=SL1.SS1.IF2.ST5, InterfaceType=Powerlink, Type=ncV_AXIS, Channel=2, Disabled=TRUE, ModuleDisabled=FALSE)
  NcObject Axis1 (ModuleAddress=SL1.SS1.IF2.ST1, InterfaceType=Powerlink, Type=ncAXIS, Channel=1, InitParameter=A1_Init, AcoposParameter=A1_Par, Disabled=FALSE, ModuleDisabled=FALSE)
  NcObject SL1.SS1.IF2.ST1.VAxis1 (ModuleAddress=SL1.SS1.IF2.ST1, InterfaceType=Powerlink, Type=ncV_AXIS, Channel=1, Disabled=FALSE, ModuleDisabled=FALSE)
  NcObject SL1.SS1.IF2.ST1.Axis2 (ModuleAddress=SL1.SS1.IF2.ST1, InterfaceType=Powerlink, Type=ncAXIS, Channel=2, Disabled=FALSE, ModuleDisabled=FALSE)
  NcObject Axis11 (ModuleAddress=SL1.SS1.IF2.ST1, InterfaceType=Powerlink, Type=ncV_AXIS, Channel=2, InitParameter=A11_Init, AcoposParameter=A11_Par, Disabled=FALSE, ModuleDisabled=FALSE)
  NcObject Axis0 (ModuleAddress=SL1.SS1.IF2.ST10, InterfaceType=Powerlink, Type=ncAXIS, Channel=1, InitParameter=A0_Init, AcoposParameter=A0_Par, Disabled=FALSE, ModuleDisabled=FALSE)
  NcObject SL1.SS1.IF2.ST10.VAxis1 (ModuleAddress=SL1.SS1.IF2.ST10, InterfaceType=Powerlink, Type=ncV_AXIS, Channel=1, Disabled=TRUE, ModuleDisabled=FALSE)
  NcObject SL1.SS1.IF2.ST10.Axis2 (ModuleAddress=SL1.SS1.IF2.ST10, InterfaceType=Powerlink, Type=ncAXIS, Channel=2, Disabled=FALSE, ModuleDisabled=FALSE)
  NcObject SL1.SS1.IF2.ST10.VAxis2 (ModuleAddress=SL1.SS1.IF2.ST10, InterfaceType=Powerlink, Type=ncV_AXIS, Channel=2, Disabled=TRUE, ModuleDisabled=FALSE)
  NcObject SL1.SS1.IF2.ST2.Axis2 (ModuleAddress=SL1.SS1.IF2.ST2, InterfaceType=Powerlink, Type=ncAXIS, Channel=2, Disabled=FALSE, ModuleDisabled=FALSE)
  NcObject SL1.SS1.IF2.ST2.VAxis2 (ModuleAddress=SL1.SS1.IF2.ST2, InterfaceType=Powerlink, Type=ncV_AXIS, Channel=2, Disabled=TRUE, ModuleDisabled=FALSE)
  NcObject Axis2 (ModuleAddress=SL1.SS1.IF2.ST2, InterfaceType=Powerlink, Type=ncAXIS, Channel=1, InitParameter=A2_Init, AcoposParameter=A2_Par, Disabled=FALSE, ModuleDisabled=FALSE)
  NcObject SL1.SS1.IF2.ST2.VAxis1 (ModuleAddress=SL1.SS1.IF2.ST2, InterfaceType=Powerlink, Type=ncV_AXIS, Channel=1, Disabled=TRUE, ModuleDisabled=FALSE)
  NcObject Axis7 (ModuleAddress=SL1.SS1.IF2.ST7, InterfaceType=Powerlink, Type=ncAXIS, Channel=1, InitParameter=A7_Init, AcoposParameter=A7_Par, Disabled=FALSE, ModuleDisabled=FALSE)
  NcObject SL1.SS1.IF2.ST7.VAxis1 (ModuleAddress=SL1.SS1.IF2.ST7, InterfaceType=Powerlink, Type=ncV_AXIS, Channel=1, Disabled=TRUE, ModuleDisabled=FALSE)
  NcObject SL1.SS1.IF2.ST7.Axis2 (ModuleAddress=SL1.SS1.IF2.ST7, InterfaceType=Powerlink, Type=ncAXIS, Channel=2, Disabled=FALSE, ModuleDisabled=FALSE)
  NcObject SL1.SS1.IF2.ST7.VAxis2 (ModuleAddress=SL1.SS1.IF2.ST7, InterfaceType=Powerlink, Type=ncV_AXIS, Channel=2, Disabled=TRUE, ModuleDisabled=FALSE)
```

## Configuration Simul_AR000

CPU , AutomationRuntime F3.01, Build 4.1.1, Vc V3.64.2

### Task classes (Cpu.sw)
```
Cyclic#1 (cycle 10000 us, tolerance 0 us):
  A9_Basic <- BagMachine_Section.MasterAxis.A9_Init.A9_Basic.prg
  A9_Control <- BagMachine_Section.MasterAxis.A9_Init.A9_Control.prg
  A15_Basic <- BagMachine_Section.HotMicroPerf.Axis15.A15_Basic.prg
  A15_Automa <- BagMachine_Section.HotMicroPerf.Axis15.A15_Automat.prg
Cyclic#4 (cycle 1000000 us, tolerance 10000000 us):
  A15_Contro <- BagMachine_Section.HotMicroPerf.Axis15.A15_Control.prg
  A15_Motion <- BagMachine_Section.HotMicroPerf.Axis15.A15_MotionCycle.prg
  HMPerf_Gen <- BagMachine_Section.HotMicroPerf.HMPerf_Gen.prg
  Test_Simul <- BagMachine_Section.BagBundler.Test_Simul.prg
DataObjects: arsdmsvp, arsdmsvg, arsdmhtm, Acp10sys
NcDataObjects: A9_Par <- BagMachine_Section.MasterAxis.A9_Init.A9_Par.dob, A15_Init <- BagMachine_Section.HotMicroPerf.Axis15.A15_Init.dob, A15_Par <- BagMachine_Section.HotMicroPerf.Axis15.A15_Par.dob, A9_Init <- BagMachine_Section.MasterAxis.A9_Init.A9_Init.dob, A1_Par, A1_Init, Config1_SL <- Config1_SL1_SS1_IF2_ST2_M1.dob, Config1_S1 <- Config1_SL1_SS1_IF2_ST10_SS2.dob
Binaries: arsdm, webserv, Acp10map, ashwd, sysconf, arconfig, iomap, asfw, Acp10cfg, vccnum, vcnet, HMI_10, HMI_1003, vcpdvnc, vcbclass, vcgclass, vccbtn, vcpfar00, vcshared, vccline, vccdt, vcalarm, vccddbox, vcfntttf, arialbd, vctcal, vccovl, vcdsloc, visvc, vccbmp, arial, vcpdsw, vcdsint, vcfile, vccshape, HMI_1001, vcmgr, vcresman, vccstr, visapi, vcchspot, vccpopup, vcrt, HMI_1002, arialbi, vcctext, vcclbox, vccalarm
Libraries: Brsystem, NcGlobal, HGWeber, astime, runtime, powerlnk, Acp10sdc, Acp10man, Acp10par, fileio, sys_lib, asmem, standard, convert, dataobj, astcp, Acp10_MC
```

### Hardware
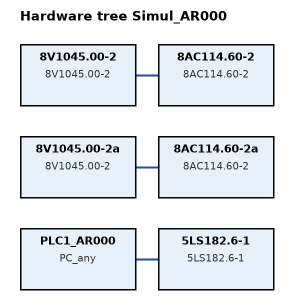
```
5LS182.6-1 : 5LS182.6-1 v1.3.1.0  [SL -> PLC1_AR000.SL1]
  Connector IF1:
    DNAConfiguration = manual
8AC114.60-2 : 8AC114.60-2 v1.0.0.8  [SS -> 8V1045.00-2.SS1; PLK1 -> 5LS182.6-1.IF1 (NodeNumber=1) [Cable Type=PowerlinkCable, Length=10, Version=1.0.0.3]; PLK2 -> 8AC114.60-2a.PLK1 (NodeNumber=1) [Cable Type=PowerlinkCable, Length=10, Version=1.0.0.3]]
8AC114.60-2a : 8AC114.60-2 v1.0.0.8  [SS -> 8V1045.00-2a.SS1; PLK1 -> 8AC114.60-2.PLK2 (NodeNumber=2) [Cable Type=PowerlinkCable, Length=10, Version=1.0.0.3]]
8V1045.00-2 : 8V1045.00-2 v2.2.0.0
  Simulate = standard
8V1045.00-2a : 8V1045.00-2 v2.2.0.0
  Simulate = standard
PLC1_AR000 : PC_any v1.1.1.0 (OrderNumber=PC)
  Connector IF3:
    Vnc1
    VncVcObjectName1 = HMI_10
    VncPortNumber1 = 5900
    VncMaxConnections1 = 1
    VncRefreshRate1 = 1000
    VncConnectionTimeout1 = 4
  VolatileGlobalPvSize = 20000
  XLinkUseDefault = 0
  Cyclic1Duration = 10000
  Cyclic1Tolerance = 0
  Cyclic1Output = 1
  Cyclic2Duration = 200000
  Cyclic2Tolerance = 10000000
  Cyclic3Duration = 500000
  Cyclic3Tolerance = 10000000
  Cyclic4Duration = 1000000
  Cyclic4Tolerance = 10000000
  Cyclic5Duration = 2000000
  Cyclic5Tolerance = 10000000
  Cyclic6Duration = 3000000
  Cyclic6Tolerance = 12000000
  Cyclic7Duration = 4000000
  Cyclic7Tolerance = 12000000
  Cyclic8Duration = 5000000
  Cyclic8Tolerance = 30000000
  TransferWebServ = 1
  TransferArSdm = 1
  TransferArSdmSvg = 1
  TransferArSdmSvp = 1
  TransferArSdmHtm = 1
```

### Acp10cfg.ncc - PLC1_AR000/Motion/Acp10cfg.ncc
```
NcConfiguration (Version=2.24.0, NcSwId=acp10)
  ACP10CF1_typ:
    cnt_nettrc_rec_drive = 1500
    bufsize_trace_upload = 1200
    tc_nc_man_task = Cyclic #1
    glob_pv_as_ncobject = Yes
    network_init:
      ncsw_init_execute = Yes
      automatic_execute = No
      node_nr_warning = Yes
      net_err_before_ncact = Yes
    nettrc:
      enter_parsecrec = Yes
      enter_ncaction = Yes
      save_ring_startidx = Yes
    sdc_if[0]:
      if_name = SDC_IF1
      mc_broadcast_size = 800
```

### Acp10map.ncm - PLC1_AR000/Motion/Acp10map.ncm
```
NcMapping (NcSwId=acp10)
  NcObject Axis9 (ModuleAddress=SDC_IF1.ST1, InterfaceType=SDC, Type=ncAXIS, Channel=1, InitParameter=A9_Init, AcoposParameter=A9_Par, Disabled=FALSE, ModuleDisabled=FALSE)
  NcObject Axis15 (ModuleAddress=SDC_IF1.ST2, InterfaceType=SDC, Type=ncAXIS, Channel=1, InitParameter=A15_Init, AcoposParameter=A15_Par, Disabled=FALSE, ModuleDisabled=FALSE)
```

## Logical view

Binary libraries used (declarations not repeated): Convert, Runtime, Operator, Brsystem, AsMath, asstring, astime, FileIO, powerlnk, AsMem, AsIOAcc, Visapi, AsARCfg, standard, sys_lib, Acp10sdc 2.24.0, NcGlobal 0.60.3, Acp10man 2.24.0, Acp10par 2.24.0, Acp10_MC 2.24.0, LoopConR

### Program Logical/Information (IEC) - A new program

#### InformationCyclic.st
```iecst
(********************************************************************
 * COPYRIGHT -- .
 ********************************************************************
 * Program: Information
 * File: InformationCyclic.st
 * Author: dominique
 * Created: October 29, 2011
 ********************************************************************
 * Implementation of program Information
 ********************************************************************)

PROGRAM _CYCLIC
  (*

    D.M. Le 04/13/2012  Pyrollpack_14661    Version programme Mise a jour apres livraison

    Reste a valider :
    --------------------------------------------
      1) Decalage dep manu Axes Arra + TE + ApPo + ArraPo
         --> A l'arret : Dep Manu
         --> En marche : Dep Manu + Calage Offset

      2) Decalage Perfo en marche

      3) Resynchro des axes
         --> Cas 4 pinces sac normal
         --> Cas 2 pinces sac normal
         --> Cas sac Pochette

      4) Position Axe ApPo en position de mainiten
         --> Cas sac normal
         --> Cas sac Pochette
         corriger le cas echeant la valeur du parametre "gr_rPosEnvBHoldBag"

      5) Calcul temoin ApPo en zone de contacte

    Pyrollpack_14661

    Perf               : 8LSC5B.E1030D005-0     F8LSC5BE103
    EntryPull_ExitPull : 8LSA73.E0030D100-0     F8LSA73E003A
    Holding_Tearing    : 8LSA73.EB030D100-0     F8LSA73EB03
    Drum               : 8LSA73.EB030D100-0     F8LSA73EB03
    IF                 : 1PH7 137-2ED03-0CA3    FPH71372ED03   (Codeur Abs EnDat Multitour)

  //------------------------------------------------------------------------------------------------------------------
    // Synchro ratio with Virtual Master

    Case Normal Bag production
    ------------------------------
    Tube length | Holding | Tearing | Env Bag | Tear EB | Drum
   --------------------------------------------------------------
    [160, 400]  |   1/2   |    1    |   1/4   |    1    |   1
   --------------------------------------------------------------
    ]400, 500]  |    1    |    2    |   1/2   |    2    |   2
   --------------------------------------------------------------
    ]500, 760]  |    1    |    2    |   1/2   |    2    |   2

    Case Envelope Bag production
    ------------------------------
    Tube length | Holding | Tearing | Env Bag | Tear EB | Drum
   --------------------------------------------------------------
    [260, 320[  |   1/2   |    2    |   1     |    2    |   2
   --------------------------------------------------------------
    ]320, 760]  |    1    |    2    |   1     |    2    |   2

    D.M. Le 07/11/2011  BrownPaper_14606

Fonctions Validees :

Fonctions encore a implementer ou finir :

    Reste a faire
    --------------------------------------------
      1) Sechage IF
         CODE     => Regul Chauffe (Finalement faite par regualtion externe cause pas le temps de developper un programme)
         CODE     => Bat TOR
         CODE     => Defaut Thermostat secu + moteurs Soufflage + batterie chauffe + Defaut sonde temperarure (arret chauffe)
         => ATENTION Codage Ok mais Reste a etre valide

      2) WISTA
         OK       => Gestion Axe
         => Synchro Axe avec conservation de offset
         => Passage de Synchro a RL et vis et versa
         => Calage en marche + ecran + commutateurs sur appareil (depuis ecran est plus pratique)
         => Du fait de RL calage a l'arret pas necessaire
         OK       => Defauts Axes
         OK       => Defaut casse bande
         OK       => Defaut carter
         OK       => Info AU

      3) Devieur bande
         OK       => Colle En/Hors
         OK       => Asservissement debit vitesse
         OK       => Soufflage En/Hors
         OK       => Defaut fin bobine Poly
         OK       => Defaut disjoncteur soufflage
         OK       => Defaut carter
         OK       => Info AU

      4) Micro Perfo a froid
         OK       => Gestion Axe
         OK       => Defauts Axes
         OK       => Defaut disjoncteur aspiration dechets
         OK       => Defaut carter

         OK             5) ATTENTION   INIT DES AXES ARRA+MAIN+TE  A FAIRE + DEFINITION POSITIONS PARTICULUIERES DES AXES => REPRENDRE MEME CHOSE QUE SUR B&H

         OK             6) Rentrer config IP Client

         OK + correction Bug 7) ATTENTION AI SHUNTE PROVISOIREMENT DEFAUT PORTES IF !!!!! VOIR ALARME 70

         OK       8) ATTENTION AI INHIBE CALCUL DE DEFAUT DES MODULES I/O A METTRE A JOUR ET A REACTIVER

         OK       9) Mettre a jour nom des disjoncteurs moteur, chauffe, etc...

         OK       10) AU AXES MACHINE A L'ARRET

         OK       11) Integrer vue cadence Perfo Type 1 et 2 speciale pour RS26 (Si possible corriger vue de RS15 Cas Inch cause manque les decimales sur axe de ordonnees)

         OK       12) IHM mettre a jour I/O dans Maintenance

         OK       13) ATTENTION !!!! Decalage a l'arret Flexo fonctionne apparemment mais apres pas possible de tourner cause Flexo est beaucoup trop lente => casse la bande au niveau de AppE RS !!!  => Certainement Came Automate est reste dans Etat 4 (exactement ca)

         OK       14) ATTENTION !!!! d'apres Georges Mathe Hors Imp FP Auto sur seuil vitesse ne fonctionne pas !!!! fait Hors Imp que une x arrive a vitesse nulle
         En fait ca fonctionnait tres bien

      15) ATTENTION !!!! Calage sur Hot Micro Perf n'est pas conserve au redemarrage meme apres arret normal

         OK       16) Vue registration => ajout 1 deciamle a la valeur de correction cause comme le + souvent est <= 1   => ca affiche toujours 0 ... et on a l'impression que ca ne corrige pas

         OK       17) ATTENTION !!! Bug dans redef pos Axe Arra il ne faut pas affecter de position > au modulo => Fonction Home fait un defaut

       18) VALIDER REDEFINITION POSITION ARRA LORS DE PASSAGE 4 <--> 2 PINCES !!!!

//-----------------------------------------------------------------------------------------------------------------------------------------------
      // Modifs apportees au programme precedent

      1) Dans module programme gestion colle sur derouleur, ajout gestion colle sur guide bande => changement nom de Unw_Glue => Unw_3W_Glue

      2) Ai verouille calcul affichage ecran config Arr/MAin/TE tant que demarrage ecran non termine

      3) Ajout condition pas(AU) sur sortie Glue !!!

      4) ATTENTION !!! Bug Phasing Axes =>  Phasing_1 fait défaut lorsque dep manu axe a l'arret avec Phasing_0 => retarder la reactivation de Phasing_1 a la fin de Phasing_0

      5) ATTENTION !!! Mettre a jour calcul temoin "gGuardsOK" dans Guard_Mon

      6) ATTENTION !!! filtrer defaut carter Gates IF avec mode reglage + Modifier de telle sorte que le mode reglage n'acquitte pas autoamtiquement le defaut

      7) ATTENTION !!! Ai deplace les variables ci-dessous de Init A9_Basic --> Cyclic Setup cause lors de chargement en RUN il est arrive que ces valeurs soient remise a 0 => Passage en SERV de CPU en pleinne demonstartion client ...

                    // General parameter init
                    gr_rMachMaxSpeed_BPM := 1000.0 ;

                    // Machie Type
                    g_iMachType := C_iRS26 ;

                    // Bag size limite
                    g_rMaxBagSize_RS15_mm := 400.0 ;
                    g_rMinBagSize_RS15_mm := 105.0 ;
                    g_rMaxBagSize_RS26_mm := 760.0 ;
                    g_rMinBagSize_RS26_mm := 160.0 ;

      8) ATTENTION !!! filtrer defaut carter Gates IF avec mode reglage

      9) ATTENTION !!! ajout d'un temoin AlimPuis retarde pour calcul defaut 230V et Disjoncteur Fan Perfo cause faisait encore le defaut a la mise sous puissance

      10) Ai corrige fonction redefinition position Arra lors de passage 4 <--> 2 pinces pour limiter nouvelle position <= Modulo sinon fonction Home fait un defaut 29225

      11) Completer defaut AU a l'arret avec AxeIF

      12) Mise a jour Message 2 => Carters !!! + Axes non pret

      13) Refait vue Cad Max Perfo RS15 Inch avec decimale sur Axe des ordonnees

//*********************************************************************************************************************************************************************************

    D.M. Le 29/10/2011  B&H_14541 Programme Dev basee sur version en cours sur machine au 28/10/2011 en fin de journee (B&H_14541 Provient de programme Brown_Paper_14542)
    Ajout de :

Validation
    OK    1) Animation sur ecran en phase de synchro des Axes.

    OK    2) Modification gestion presseur AppS et IF pour eviter mise sous pression automatique sur acquittement defaut AU ou mise sous puissance.
    OK       Presseur AppE pour interdire On si BP Off active

    OK    3) Ajout courbes cadence Max machine RS26 Perfo 400mm uniquement

    OK    4) Fermeture auto affichage courbes de cadence Max machine sur sortie de la vue SetUp Perfo

    OK    5) Calage manu Perfo a l'arret

    OK    6) Calage manu IF a l'arret

    OK    7) Supression "shuntage" defaut carter

    OK    8) !!! ATTENTION !!!  Ajout d'un AU sur les axes pour le cas deplacement manu des axes machine a l'arret
    OK       + Ajout disable Axes en fin d'AU

    OK    9) Limitation a RS15 uniquement de correction position arret machine avec Arra hors position d'arrachement
    OK    + Limitation a RS15 uniquement de coupure Enable Drive Drum lorsque Home Tearing et vis et versa
    OK    + Table A4_Init Homing regalge parametres ci-dessous sur ncNEGATIVE au lieu de ncPOSITIVE pour referencement dans sens negatif
                                                  edge_sw   --> ncNEGATIVE    Edge of reference switch
                                                  start_dir --> ncNEGATIVE    Start direction
                                                  trigg_dir --> ncNEGATIVE    Trigger directionpour direction Home sens negatif conforme a RS26

    OK    10) Ajout calcul temoin "Drum in contact zone with blade" arbitrairement fixe a 20°

    OK    11) En marche calage RS sur impression

    OK    12) Correction resynchro Holding apres manu => toujours retour en Etat 2 (Synchro OK) puisque axe vient d'etre regle en manu !!! => donc il faut conserver ce reglage !!!

    OK    13) Decomposition decalage Offset Drum en marche

    OK    14) Adaptation position de Reference Tearing Axis en fonction du Format (+/-180° cas 2 pinces a voir) + adapattion cycle referencement cas RS26 ou RS15

    OK    15) Ai ajouter filtre selection DHS pour prod sur affichage message deselection fin de bobines DHS

    OK    16) Modif defaut 230V pour que fasse defaut uniquement lorsque PowerOn et pas entree 230V active

    OK    17) Modif calcul defaut disjoncteur Fan Perfo pour que fasse defaut que si Ligne 24V pas coupee (Power On , pas AU pas def Carter, etc...)

    OK    18) Correction Beug Action Etape6 venant de Etape2 cycle manu Main => ajouter : "gstCycA[3].CycManTimSet.CmdSynchroOn := 0 ;"

    OK    19) Réglage de tous les Offsets de referencemet à 0°

    OK    20) Ajout position caracreristiques de axeq Arra Main et TE lorsque Arra arrache (est a la vertical) Main maintien (est a la vertical) et pince tambour pince le sac (Lame dans la pince)

    OK    21) Position init des axes Main + Arra + TE => Pour simplifier parametrage ai mis le meme offset sur les 3 Axes = 20°

    OK    22) Corriger I/0 dans vues maintenance

    OK    23) Corriger cad max Perfo points particuliers transition 1 <--> 2 Perfo

    OK    24) Demande auto operateur positionner Holding+Tearinf+Drum axis dans config correcte lors de passage 4 <--> 2 pinces
       OK =>  + Verifier si toujours possible d'aboutir a la config demandee
       OK =>  + Si trop complique demander a operateur de positionner stations conformement a image sur IHM et de confirmer par un boutton => redefinir position correcte de Arra et Maint

    OK    25) Mise a jour recettage

    Reste a faire
    --------------------------------------------

    ??) Modulation tension de bande AppE en fonction de VL

    ATTENTION !!!! A FAIRE AVANT DEPART MACHINE

    OK    1) Config IP client a rentrer

      2) Niveau Bus DC Puis a adapte pour tension client Udc = Racive(2)*Ueff = 480 x 1.414 = 678.82 V

   *)
END_PROGRAM
```

### Global.typ - Global data types
```iecst
TYPE
  PasswordLevel :   STRUCT
    Operator : STRING[32];
    Supervisor : STRING[32];
    Maintenance : STRING[32];
    Technician : STRING[32];
END_STRUCT;
  Recipe : 	STRUCT
    Name : STRING[32];
    Repeat : REAL;
    PackCount : DINT;
    HoldCount : DINT;
    Perf_Offset : REAL;
    Holding_Offset : REAL;
    Tearing_Offset : REAL;
    Drum_Offset : REAL;
    rPerf_PhasMasterDeg    : REAL;
    rHolding_PhasMasterDeg : REAL;
    rTearing_PhasMasterDeg : REAL;
    rDrum_PhasMasterDeg    : REAL;
    rCMPerf_OffsetIn       : REAL; (*Offset of the Cold Micro-Perf Axis, in Inch*)
    rCMPerf_PhasMasterDeg  : REAL; (*Phase of the Cold Micro-Perf Axis, in Deg*)
    rHMPerf_OffsetIn       : REAL; (*Offset of the Hot Micro-Perf Axis, in Inch*)
    rHMPerf_PhasMasterDeg  : REAL; (*Phase of the Hot Micro-Perf Axis, in Deg*)
    rEnvB_PhasMasterDeg    : REAL; (*Phase of the Envelope Bag Axis, in Deg*)
    rTearEB_PhasMasterDeg  : REAL; (*Phase of the Tearing Envelope Bag Axis, in Deg*)
    rEnvB_Offset           : REAL; (*Offset of the Envelope Bag Axis, in Deg*)
    rTearEB_Offset         : REAL; (*Offset of the Tearing Envelope Bag Axis, in Deg*)
    rEnvB_PerfSize_in      : REAL; (*Size = perimeter of the Envelope Bag Perforator, in Inch*)
    Entry_Draw   : REAL;
    Exit_Draw    : REAL;
    rCMPerf_Draw : REAL; (*Cold Micro Perf draw setpoint, in %*)
    bCMPerf_Mode : BOOL; (*Mode operation Cold Micro Perf, =0:Continu, =1:Interrupt*)
    rHotMicroPerfSize_in : REAL ; (*Perimeter of the tool of the Hot Micro Perf, in in*)
    bHMPerf_Mode : BOOL; (*Mode operation Hot Micro Perf, =0:Continu, =1:Interrupt*)
    iHMPerf_Up   : INT;  (*In case interrupt = Number of repeat per round on Tool*)
    bSelFPProd   : BOOL ;
    bSelHeaterProd : BOOL ;
    rHeatSPDegF : REAL ;
    bSelColdMicroPerfProd : BOOL ;
    bSelEnvBProd : BOOL ; (*Activation Envelope Bag for production =0:Off, =1:On*)
    rSlopeExitTable : REAL ;
    bSelTypeRSGlue : BOOL; (*Type RS glue selection, =0:Cold; =1:Hot*)
    bSelTypeOtherRSGlue : BOOL; (*Type Other RS glue selection, =0:Cold; =1:Hot*)
    iNumToothGearPrint : INT ; (*Number of tooth on the Gear printing repeat, in case Flexo Press*)
    iPrintUp : INT ; (*Number of picture per round on printing cylinder, in case Flexo Press*)
END_STRUCT;
  Registration : 	STRUCT
    Enable : BOOL;
    Ind_General : UINT;
    Ind_Text : UINT;
    Ind_Color : UINT;
    SP_Repeat : REAL;
    SP_MaximumCorrection : REAL;
    SP_Format : REAL;
    SP_Tolerance : REAL;
    SP_Offset : REAL;
    SP_WeightingFactor : REAL;
    SP_MarkMissedCount : DINT;
    SP_OutOfToleranceCount : DINT;
    SP_PE_Distance : REAL;
    Pointer : USINT;
    LengthActual : REAL;
    LengthAverage : REAL;
    LengthCorrection : REAL;
    OffsetActive : BOOL;
    CorrectionMax : BOOL;
    CorrectionNew : BOOL;
    MarkFirst : BOOL;
    MarkGood : BOOL;
    MarkGoodNew : BOOL;
    MarkGoodCount : DINT;
    MarkMissed : BOOL;
    MarkMissedNew : BOOL;
    MarkMissedCount : DINT;
    ShutdownMissedMark : BOOL;
    ShutdownOutOfTolerance : BOOL;
END_STRUCT;
  Encoder : 	STRUCT
    Ident : UDINT;
    Error : BOOL;
    ErrorID : UINT;
    ErrorCount : UINT;
    ErrrorText : ARRAY[0..3] OF STRING[79];
    ParID_1 : UINT;
    ParID_2 : UINT;
    ParID_1_Ready : BOOL;
    ParID_2_Ready : BOOL;
    Cmd_Reset : BOOL;
    SP_PPR : REAL;
    MachinePeriod : REAL;
    UnitsPerInch : REAL;
    UnitsPerDeg : REAL;
    PositionCount : REAL;
    PositionInch : REAL;
    PositionDeg : REAL;
END_STRUCT;
  AxisSP : 	STRUCT
    HomeOffset : REAL;
    PhaseOffset : REAL;
    Diameter : REAL;
    ParkPosition : REAL;
    MatchedSpeed : REAL;
    AbsoluteOffset : REAL;
    rZoneBefPerf_in : REAL; (*Zone matched speed before Perf, in inch*)
    rZoneAftPerf_in : REAL; (*Zone matched speed after Perf, in inch*)
END_STRUCT;
  AxisBasic : 	STRUCT
    Ident : UDINT;
    Error : BOOL;
    ErrorStop : BOOL;
    ErrorID : UINT;
    ErrorCount : UINT;
    ErrorAck : BOOL;
    ErrorText : ARRAY[0..3] OF STRING[79];
    Ind_Enabled : BOOL;
    Ind_Ready : BOOL;
    Ind_Stopping : BOOL;
    Ind_StandStill : BOOL;
    Ind_InMotion : BOOL;
    Ind_Homed : BOOL;
    Ind_Homing : BOOL;
    Ind_DiscreteMotion : BOOL;
    Ind_ContinuousMotion : BOOL;
    Ind_SynchronizedMotion : BOOL;
    Ind_AutomatEnabled : BOOL;
    Ind_CurrentAutomatState : USINT;
    Ind_Simulation : BOOL;
    Ind_NetworkInit : BOOL;
    Ind_ControllerReady : BOOL;
    Ind_ControllerStatus : BOOL;
    Ind_HomingOk : BOOL;
    Ind_LagWarning : BOOL;
    Ind_bInContactZone : BOOL; (*= 1 if Axis is in contact zone; =0 else*)
    Ind_bSynchroOK     : BOOL; (*= 1 When synchronisation with Master is finished; =0 else*)
    bSynchroReq        : BOOL; (*= 1 When synchronisation is required; =0 else*)
    Cmd_Enable : BOOL;
    Cmd_DiscreteMotion : BOOL;
    Cmd_ContinuousMotion : BOOL;
    Cmd_ContinuousMotionUpdate : BOOL;
    Cmd_SynchronizedMotion : BOOL;
    Cmd_SynchronizedMotionUpdate : BOOL;
    Cmd_PhaseOffset : BOOL;
    Cmd_Halt : BOOL;
    iPhasingState : INT ; (*Phasing command actual state : =0:rest; =1:busy; =2:Error*)
    Cmd_Home : BOOL;
    Cmd_Reset : BOOL;
    Cmd_ManuTimSetPlus : BOOL;
    Cmd_ManuTimSetMinus : BOOL;
    Cmd_Override : BOOL;
    Cmd_CalcCameProf : BOOL; (*Came Profile calculation*)
    Cmd_GetMaPosProf : BOOL; (*Calculation master position in the Came Profile according to slave position*)
    Cmd_GetSlPosProf : BOOL; (*Calculation slave position in the Came Profile according to master position*)
    Cmd_EStopDisable : BOOL; (*Disable axe after EStop and machine at Standstill*)
    SP_Accel : REAL;
    SP_Decel : REAL;
    SP_EStopDecel : REAL;
    SP_GuardFaultDecel : REAL;
    SP_WebBreakDecel : REAL;
    SP_GenFaultDecel : REAL;
    SP_FStopDecel : REAL;
    SP_JogDecel : REAL;
    SP_Velocity : REAL;
    SP_Distance : REAL;
    SP_PhaseOffset : REAL;
    SP_GearBoxInput : REAL;
    SP_GearBoxOutput : REAL;
    SP_MotorPPR : REAL;
    rSP_OverrideV : REAL;
    rSP_OverrideA : REAL;
    rSP_CorPosVel : REAL ; (*Position correction according to the speed because of dead time and in order to match with the virtual master position, in °/rpm*)
    rSP_Pos_Deg : REAL ;   (*Input set point position of the position controller ParID 428, in deg*)
    rPerim_In   : REAL ;   (*Perimeter of the Axis, in inch*)
    bActive     : BOOL ;   (*Axis activated*)
    bInMach     : BOOL ;   (*Axis in machine, =0:NO, =1:YES*)
    HomeVelocity : REAL;
    PositionCount : REAL;
    PositionInch : REAL;
    PositionDeg : REAL;
    rSetPosCount : REAL;
    rSetPosInch : REAL;
    rSetPosDeg : REAL;
    rActPhasDeg : REAL; (*Calculated actual Master/Slave Phase; PosSlave = RatioSynchro*PosMaster + Phase, in Deg*)
    rRSynNum : REAL; (*Sychro ratio numerator Master/Slave, PosSlave = RatioSynchro*PosMaster + Phase,  RatioSynchro = rRSynNum/rRSynDen*)
    rRSynDen : REAL; (*Sychro ratio denominator Master/Slave, PosSlave = RatioSynchro*PosMaster + Phase,  RatioSynchro = rRSynNum/rRSynDen*)
    uiiNumRev : UDINT ; (*Number of revolution*)
    AxisPeriod : REAL;
    ActualVelocity : REAL;
    ActualTorque : REAL;
    UnitsPerInch : REAL;
    UnitsPerDeg : REAL;
    InchPerDeg : REAL;
    Input_Home : BOOL;
    Input_PosHW : BOOL;
    Input_NegHW : BOOL;
    Input_Trigger1 : BOOL;
    Input_Trigger2 : BOOL;
    Input_DriveEnable : BOOL;
END_STRUCT;
  RECIPE_CNTL_typ : 	STRUCT
    cmdDelete : BOOL;
    cmdLoad : BOOL;
    cmdSave : BOOL;
    currRecipe : STRING[20];
    description : STRING[80];
    driveSelect : USINT;
    newRecipe : STRING[20];
    opActive : BOOL;
    status : STRING[40];
END_STRUCT;
  RECIPE_typ : 	STRUCT
    description : STRING[80];
    dataDINT : ARRAY[0..9] OF DINT;
    dataReal : ARRAY[0..9] OF REAL;
    dataCheck : DINT;
END_STRUCT;
  System : 	STRUCT
    gSP_A : ARRAY[0..15] OF AxisSP;
    gReg : ARRAY[0..15] OF Registration;
    gPassword : PasswordLevel;
    gMachineTime : HourMeter;
    gSP_CmdSpeed : REAL;
    gSP_ColdGlue : Glue;
    gSP_HotGlue : Glue;
    gSP_GlueTrayAutoSpeed : REAL;
    gSP_PerfCylSelect : BOOL;
    gSP_PerfKnifeCount : REAL;
    gSP_TubeSelect : BOOL;
END_STRUCT;
  HourMeter : 	STRUCT
    Seconds : INT;
    Minutes : INT;
    Hours : DINT;
END_STRUCT;
  Glue :   STRUCT
    Start : ARRAY[0..15] OF REAL;
    Length : ARRAY[0..15] OF REAL;
    OnComp : UDINT;
    OffComp : UDINT;
    Hysteresis : REAL;
    MinPressure : REAL;
    MaxPressure : REAL;
    ManPressure : REAL;
    AutoOnSpeed : REAL;
END_STRUCT;
END_TYPE
```

### Package Logical/Cycles - A package of related programs and data objects.

### GenCycles.var
```iecst
(********************************************************************
 * COPYRIGHT -- .
 ********************************************************************
 * Package: NewPackage
 * File: NewPackage.var
 * Author: dominique
 * Created: August 01, 2011
 ********************************************************************
 * Variables of package NewPackage
 ********************************************************************

 C_iSTEP_ : Num step for cycle *)

VAR
    gstCycA : ARRAY [0..15] OF stCycAxis ;
    g_rCycManTimSetOverrideAcc : REAL ;
END_VAR

VAR CONSTANT
    C_iSTEP_0  : INT := 0 ;
    C_iSTEP_1  : INT := 1 ;
    C_iSTEP_2  : INT := 2 ;
    C_iSTEP_3  : INT := 3 ;
    C_iSTEP_4  : INT := 4 ;
    C_iSTEP_5  : INT := 5 ;
    C_iSTEP_6  : INT := 6 ;
    C_iSTEP_7  : INT := 7 ;
    C_iSTEP_8  : INT := 8 ;
    C_iSTEP_9  : INT := 9 ;
    C_iSTEP_10 : INT := 10 ;
    C_iSTEP_11 : INT := 11 ;
    C_iSTEP_12 : INT := 12 ;
    C_iSTEP_13 : INT := 13 ;
    C_iSTEP_14 : INT := 14 ;
    C_iSTEP_15 : INT := 15 ;
    C_iSTEP_16 : INT := 16 ;
    C_iSTEP_17 : INT := 17 ;
    C_iSTEP_18 : INT := 18 ;
    C_iSTEP_19 : INT := 19 ;
    C_iSTEP_20 : INT := 20 ;
    C_iSTEP_21 : INT := 21 ;
    C_iSTEP_22 : INT := 22 ;
    C_iSTEP_23 : INT := 23 ;
    C_iSTEP_24 : INT := 24 ;
    C_iSTEP_25 : INT := 25 ;
    C_iSTEP_26 : INT := 26 ;
    C_iSTEP_27 : INT := 27 ;
    C_iSTEP_28 : INT := 28 ;
    C_iSTEP_29 : INT := 29 ;
    C_iSTEP_30 : INT := 30 ;
    C_iSTEP_31 : INT := 31 ;
    C_iSTEP_32 : INT := 32 ;
    C_iSTEP_33 : INT := 33 ;
    C_iSTEP_34 : INT := 34 ;
    C_iSTEP_35 : INT := 35 ;
    C_iSTEP_36 : INT := 36 ;
    C_iSTEP_37 : INT := 37 ;
    C_iSTEP_38 : INT := 38 ;
    C_iSTEP_39 : INT := 39 ;
    C_iSTEP_40 : INT := 40 ;
    C_iSTEP_41 : INT := 41 ;
    C_iSTEP_42 : INT := 42 ;
    C_iSTEP_43 : INT := 43 ;
    C_iSTEP_44 : INT := 44 ;
    C_iSTEP_45 : INT := 45 ;
    C_iSTEP_46 : INT := 46 ;
    C_iSTEP_47 : INT := 47 ;
    C_iSTEP_48 : INT := 48 ;
    C_iSTEP_49 : INT := 49 ;
    C_iSTEP_99 : INT := 99 ;
END_VAR
```

### Package Logical/Libraries - Global libraries

### Library Logical/Libraries/HGWeber (IEC) - HG Weber Function Blocks

#### H_FB_2StepMove.st
```iecst
(********************************************************************
 * COPYRIGHT --

 ********************************************************************
 * Library: HGWeber
 * File: H_FB_2StepMove.st
 * Author: dominique
 * Created: August 18, 2011
 ********************************************************************
 * Implementation of library HGWeber
 ********************************************************************)

(* TODO: Add your comment here *)
FUNCTION_BLOCK H_FB_2StepMove

  IF EDGEPOS(IN_bStart) AND
     IN_bPermis         AND
     ( iStep = 0 )      THEN
    iStep := 1 ;
    RETURN ;
  END_IF

  IF NOT(IN_bPermis) THEN
    iStep          := 0 ;
    OUT_bHorn      := 0 ;
    OUT_bStartMove := 0 ;

  END_IF

  stTON_0(IN:=(iStep=1), PT:=IN_tTpHorn) ;
  stTON_1(IN:=(iStep=2), PT:=T#2s) ;
  stTON_2(IN:=(iStep=3), PT:=T#2s) ;
  stTON_3(IN:=(iStep=4), PT:=T#1s) ;

  CASE iStep OF
    1 : ; // Horn ringing
        IF IN_bStart THEN
          OUT_bHorn := 1 ;
          IF stTON_0.Q THEN
            iStep     := 2 ;
            OUT_bHorn := 0 ;
          END_IF
        ELSE
          iStep     := 0 ;
          OUT_bHorn := 0 ;
        END_IF
    2 : ; // Waiting remove start
        IF NOT(stTON_1.Q) THEN
          IF NOT(IN_bStart) THEN
            iStep := 3 ;
          END_IF
        ELSE
          iStep := 0 ;
        END_IF
    3 : ; // Waiting new start
        IF NOT(stTON_2.Q) THEN
          IF IN_bStart THEN
            iStep := 4 ;
            OUT_bStartMove := 1 ;
          END_IF
        ELSE
          iStep := 0 ;
        END_IF
    4 : ; // Output during 1s
        IF stTON_3.Q THEN
          iStep := 0 ;
          OUT_bStartMove := 0 ;
        END_IF
  END_CASE
  OUT_iActStep := iStep ;
END_FUNCTION_BLOCK
```

#### H_FB_ToggleTB.st
```iecst
(********************************************************************
 * COPYRIGHT -- .
 ********************************************************************
 * Library: HGWeber
 * File: H_FB_ToggleTB.st
 * Author: dominique
 * Created: August 19, 2011
 ********************************************************************
 * Implementation of library HGWeber
 ********************************************************************)

FUNCTION_BLOCK H_FB_ToggleTB

    IF IN_bTB THEN
      OUT_uiTxt_Ind := IN_uiTxt1_Ind ;
    ELSE
      OUT_uiTxt_Ind := IN_uiTxt0_Ind ;
    END_IF

    IF IN_bTB THEN
      OUT_uiCol_Ind := IN_uiBackCol_State0 + IN_uiForeCol_State0 * 256;
    ELSE
      OUT_uiCol_Ind := IN_uiBackCol_State1 + IN_uiForeCol_State1 * 256;
    END_IF

END_FUNCTION_BLOCK
```

#### H_FB_WatchSensor.st
```iecst
(********************************************************************
 * COPYRIGHT -- .
 ********************************************************************
 * Library: HGWeber
 * File: H_FB_WatchSensor.st
 * Author: dominique
 * Created: August 19, 2011
 ********************************************************************
 * Implementation of library HGWeber
 ********************************************************************)

FUNCTION_BLOCK H_FB_WatchSensor
    // Reset fault
    bReset := EDGEPOS(IN_bReset) ;
    // Filtering sensor input
    stTON_FiltSensIn(IN:=IN_bSensorIn, PT:=IN_tTpFiltDI);
    stTON_FiltSensOut(IN:=IN_bSensorOut, PT:=IN_tTpFiltDI);
    stTOF_FiltSensIn(IN:=stTON_FiltSensIn.Q, PT:=IN_tTpFiltDI) ;
    stTOF_FiltSensOut(IN:=stTON_FiltSensOut.Q, PT:=IN_tTpFiltDI) ;

    bSensorIn  := stTOF_FiltSensIn.Q ;
    bSensorOut := stTOF_FiltSensOut.Q ;

    // Fault calculation
    stTON_SOL_Out(IN:=IN_bSOL_Out AND NOT(bReset), PT:=IN_tTpWatchOut+IN_tTpFiltDI) ;
    stTON_SOL_In(IN:=IN_bSOL_In AND NOT(bReset), PT:=IN_tTpWatchIn+IN_tTpFiltDI) ;
    IF stTON_SOL_Out.Q THEN
      IF bSensorIn THEN
        OUT_bSensIn_FaultOut := IN_bActSensIn ;
      END_IF
      IF NOT(bSensorOut) THEN
        OUT_bSensOut_FaultOut := IN_bActSensOut ;
      END_IF
    END_IF

    IF stTON_SOL_In.Q THEN
      IF NOT(bSensorIn) THEN
        OUT_bSensIn_FaultIn := IN_bActSensIn ;
      END_IF
      IF bSensorOut THEN
        OUT_bSensOut_FaultIn := IN_bActSensOut ;
      END_IF
    END_IF

    IF bReset THEN
      OUT_bSensIn_FaultOut  := 0 ;
      OUT_bSensOut_FaultOut := 0 ;
      OUT_bSensIn_FaultIn   := 0 ;
      OUT_bSensOut_FaultIn  := 0 ;
    END_IF

    OUT_bSensIn_Fault  := OUT_bSensIn_FaultOut OR OUT_bSensIn_FaultIn ;
    OUT_bSensOut_Fault := OUT_bSensOut_FaultOut OR OUT_bSensOut_FaultIn ;
    OUT_bSens_Fault    := OUT_bSensIn_Fault OR OUT_bSensOut_Fault ;

END_FUNCTION_BLOCK
```

#### H_FC_Modulus.st
```iecst
(********************************************************************
 * COPYRIGHT -- .
 ********************************************************************
 * Library: HGWeber
 * File: H_FC_Modulus.st
 * Author: dominique
 * Created: February 09, 2012
 ********************************************************************
 * Implementation of library HGWeber
 ********************************************************************)

(* TODO: Add your comment here *)
FUNCTION H_FC_Modulus(*Calculat the modulus of number*)

  IF (IN_rVar>=0.0) THEN
    rVar := IN_rVar - TRUNC(IN_rVar/IN_rMod)*IN_rMod ;
  ELSE
    rVar := IN_rVar + TRUNC(ABS(IN_rVar)/IN_rMod+1)*IN_rMod ;
  END_IF

  H_FC_Modulus := rVar ;

END_FUNCTION
```

#### H_FC_Modulus_V0.st
```iecst
(********************************************************************
 * COPYRIGHT -- .
 ********************************************************************
 * Library: HGWeber
 * File: NewFunction.st
 * Author: dominique
 * Created: August 04, 2011
 ********************************************************************
 * Implementation of library HGWeber
 ********************************************************************)

FUNCTION H_FC_Modulus_V0 (*Calculat the modulus of number*)
    rVar := IN_rVar ;

WHILE rVar < 0.0 DO
    rVar := rVar + IN_rMod ;
END_WHILE ;

WHILE rVar > IN_rMod DO
    rVar := rVar - IN_rMod ;
END_WHILE ;

H_FC_Modulus_V0 := rVar ;
END_FUNCTION
```

#### HGW_2StateIND.st
```iecst
(********************************************************************
 * COPYRIGHT --
 ********************************************************************
 * Library: HGWeber
 * File: HGW_2StateIND.st
 * Author: pkiel
 * Created: September 03, 2009
 ********************************************************************
 * Implementation of library HGWeber
 ********************************************************************)

(*Two State Indication*)
FUNCTION_BLOCK HGW_2StateIND

	IF(In_State)THEN
		Text_Ind := 1;
	ELSE
		Text_Ind := 0;
	END_IF

	CASE Text_Ind OF
		0:
			Color_Ind := BackColor_State0 + ForeColor_State0 * 256;
			State0 := 1;
			State1 := 0;
		1:
			Color_Ind := BackColor_State1 + ForeColor_State1 * 256;
			State0 := 0;
			State1 := 1;
		2:
			Text_Ind := 0;
	END_CASE

END_FUNCTION_BLOCK
```

#### HGW_2StepMove.ld
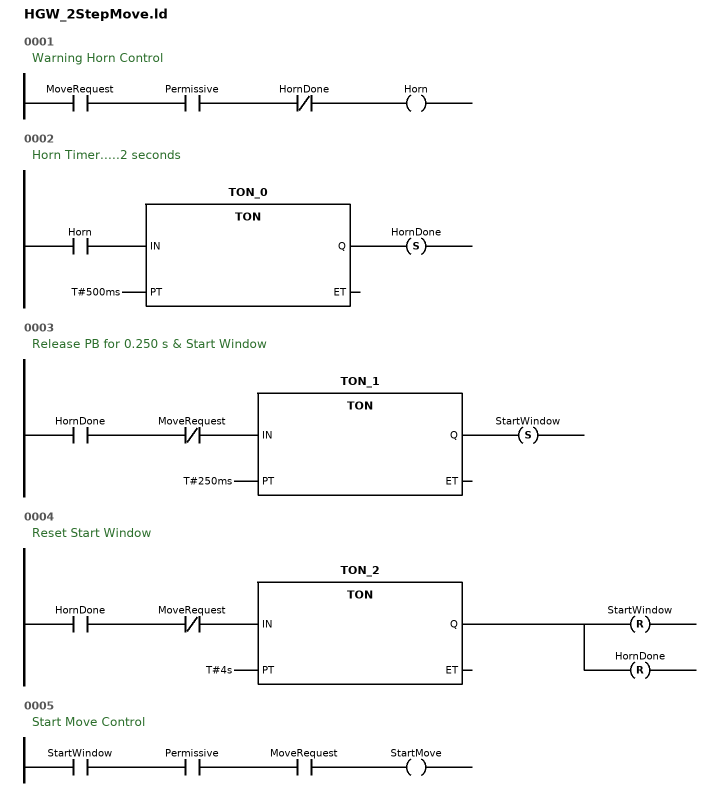
Ladder, written as Structured Text:
```iecst
FUNCTION_BLOCK HGW_2StepMove
(* Network 1: Warning Horn Control *)
Horn := MoveRequest AND Permissive AND NOT HornDone;

(* Network 2: Horn Timer.....2 seconds *)
TON_0(IN := Horn, PT := T#500ms);
IF TON_0.Q THEN HornDone := TRUE; END_IF;

(* Network 3: Release PB for 0.250 s & Start Window *)
TON_1(IN := HornDone AND NOT MoveRequest, PT := T#250ms);
IF TON_1.Q THEN StartWindow := TRUE; END_IF;

(* Network 4: Reset Start Window *)
TON_2(IN := HornDone AND NOT MoveRequest, PT := T#4s);
IF TON_2.Q THEN
    StartWindow := FALSE;
    HornDone := FALSE;
END_IF;

(* Network 5: Start Move Control *)
StartMove := StartWindow AND Permissive AND MoveRequest;
END_FUNCTION_BLOCK
```

#### HGW_3StateIND.st
```iecst
(********************************************************************
 * COPYRIGHT --
 ********************************************************************
 * Library: HGWeber
 * File: HGW_3StateIND.st
 * Author: pkiel
 * Created: September 03, 2009
 ********************************************************************
 * Implementation of library HGWeber
 ********************************************************************)

(*Three State Indication*)
FUNCTION_BLOCK HGW_3StateIND

	IF(In_State0)THEN
		Text_Ind := 0;
	END_IF
	IF(In_State1)THEN
		Text_Ind := 1;
	END_IF
	IF(In_State2)THEN
		Text_Ind := 2;
	END_IF

	CASE Text_Ind OF
		0:
			Color_Ind := BackColor_State0 + ForeColor_State0 * 256;
			State0 := 1;
			State1 := 0;
			State2 := 0;
		1:
			Color_Ind := BackColor_State1 + ForeColor_State1 * 256;
			State0 := 0;
			State1 := 1;
			State2 := 0;
		2:
			Color_Ind := BackColor_State2 + ForeColor_State2 * 256;
			State0 := 0;
			State1 := 0;
			State2 := 1;
		3:
			Text_Ind := 0;
	END_CASE

END_FUNCTION_BLOCK
```

#### HGW_3StatePB.st
```iecst
(********************************************************************
 * COPYRIGHT --
 ********************************************************************
 * Library: HGWeber
 * File: HGW_3StatePB.st
 * Author: pkiel
 * Created: September 03, 2009
 ********************************************************************
 * Implementation of library HGWeber
 ********************************************************************)

(*Three State Pushbutton Control/Indication*)
FUNCTION_BLOCK HGW_3StatePB

	R_Trig1(CLK:=PB);
	IF(R_Trig1.Q)THEN
		Text_Ind := 1 + Text_Ind;
	END_IF
	IF (Reset) THEN
		Text_Ind :=0;
	END_IF

	(* For Each Button Press, the internal state is changed...changing the text, color, and state indications *)

	CASE Text_Ind OF
		0:
			Color_Ind := BackColor_State0 + ForeColor_State0 * 256;
			State0 := 1;
			State1 := 0;
			State2 := 0;
		1:
			Color_Ind := BackColor_State1 + ForeColor_State1 * 256;
			State0 := 0;
			State1 := 1;
			State2 := 0;
		2:
			Color_Ind := BackColor_State2 + ForeColor_State2 * 256;
			State0 := 0;
			State1 := 0;
			State2 := 1;
		3:
			Text_Ind := 0;
	END_CASE

END_FUNCTION_BLOCK
```

#### HGW_4StateIND.st
```iecst
(********************************************************************
 * COPYRIGHT --
 ********************************************************************
 * Library: HGWeber
 * File: HGW_4StateIND.st
 * Author: pkiel
 * Created: September 03, 2009
 ********************************************************************
 * Implementation of library HGWeber
 ********************************************************************)

(*Four State Indication*)
FUNCTION_BLOCK HGW_4StateIND

	IF(In_State0)THEN
		Text_Ind := 0;
	END_IF
	IF(In_State1)THEN
		Text_Ind := 1;
	END_IF
	IF(In_State2)THEN
		Text_Ind := 2;
	END_IF
	IF(In_State3)THEN
		Text_Ind := 3;
	END_IF

	CASE Text_Ind OF
		0:
			Color_Ind := BackColor_State0 + ForeColor_State0 * 256;
			State0 := 1;
			State1 := 0;
			State2 := 0;
			State3 := 0;
		1:
			Color_Ind := BackColor_State1 + ForeColor_State1 * 256;
			State0 := 0;
			State1 := 1;
			State2 := 0;
			State3 := 0;
		2:
			Color_Ind := BackColor_State2 + ForeColor_State2 * 256;
			State0 := 0;
			State1 := 0;
			State2 := 1;
			State3 := 0;
		3:
			Color_Ind := BackColor_State3 + ForeColor_State3 * 256;
			State0 := 0;
			State1 := 0;
			State2 := 0;
			State3 := 1;
		4:
			Text_Ind := 0;
	END_CASE

END_FUNCTION_BLOCK
```

#### HGW_4StatePB.st
```iecst
(********************************************************************
 * COPYRIGHT --
 ********************************************************************
 * Library: HGWeber
 * File: HGW_4StatePB.st
 * Author: pkiel
 * Created: September 03, 2009
 ********************************************************************
 * Implementation of library HGWeber
 ********************************************************************)

(*Four State Pushbutton Control/Indication*)
FUNCTION_BLOCK HGW_4StatePB

	R_Trig1(CLK:=PB);
	IF(R_Trig1.Q)THEN
		Text_Ind := 1 + Text_Ind;
	END_IF
	IF (Reset) THEN
		Text_Ind :=0;
	END_IF

	(* For Each Button Press, the internal state is changed...changing the text, color, and state indications *)

	CASE Text_Ind OF
		0:
			Color_Ind := BackColor_State0 + ForeColor_State0 * 256;
			State0 := 1;
			State1 := 0;
			State2 := 0;
			State3 := 0;
		1:
			Color_Ind := BackColor_State1 + ForeColor_State1 * 256;
			State0 := 0;
			State1 := 1;
			State2 := 0;
			State3 := 0;
		2:
			Color_Ind := BackColor_State2 + ForeColor_State2 * 256;
			State0 := 0;
			State1 := 0;
			State2 := 1;
			State3 := 0;
		3:
			Color_Ind := BackColor_State3 + ForeColor_State3 * 256;
			State0 := 0;
			State1 := 0;
			State2 := 0;
			State3 := 1;
		4:
			Text_Ind := 0;
	END_CASE

END_FUNCTION_BLOCK
```

#### HGW_KeyRepeat.st
```iecst
(********************************************************************
 * COPYRIGHT --
 ********************************************************************
 * Library: HGWeber
 * File: HGW_KeyRepeat.st
 * Author: pkiel
 * Created: September 03, 2009
 ********************************************************************
 * Implementation of library HGWeber
 ********************************************************************)

(*Toggles A Bool At A Rate After An Initial Delay*)
FUNCTION_BLOCK HGW_KeyRepeat

	TON_0(IN:=Key_In,PT:=Delay);
	TON_1(IN:=(TON_0.Q AND (NOT TON_2.Q)),PT:=Rate/2);
	TON_2(IN:=TON_1.Q,PT:=Rate/2);

	R_Trig0(CLK:=Key_In);
	R_Trig1(CLK:=TON_0.Q);
	R_Trig2(CLK:=TON_1.Q);

	IF (R_Trig0.Q OR R_Trig1.Q OR R_Trig2.Q) THEN
		Key_Out:=1;
	ELSE
		Key_Out:=0;
	END_IF

END_FUNCTION_BLOCK
```

#### HGW_ScaleReal.st
```iecst
(********************************************************************
 * COPYRIGHT --
 ********************************************************************
 * Library: HGWeber
 * File: HGW_ScaleReal.st
 * Author: pkiel
 * Created: September 03, 2009
 ********************************************************************
 * Implementation of library HGWeber
 ********************************************************************)

(*Scales A Real Value A Scaled Range*)
FUNCTION_BLOCK HGW_ScaleReal

	IF (Enable) THEN
		InputDiff:=InputMax-InputMin;
		ScaledDiff:=ScaledMax-ScaledMin;
		IF (InputDiff>0) THEN
			Slope:=ScaledDiff/InputDiff;
			Offset:=ScaledMin-(InputMin*Slope);
			ScaledOut:=(InputRaw*Slope)+Offset;
			OK:=1;
			Error:=0;
		ELSE
			OK:=0;
			Error:=1;
		END_IF
	ELSE
		OK:=0;
		Error:=0;
		ScaledOut:=0;
	END_IF

END_FUNCTION_BLOCK
```

#### HGW_Toggle.ld
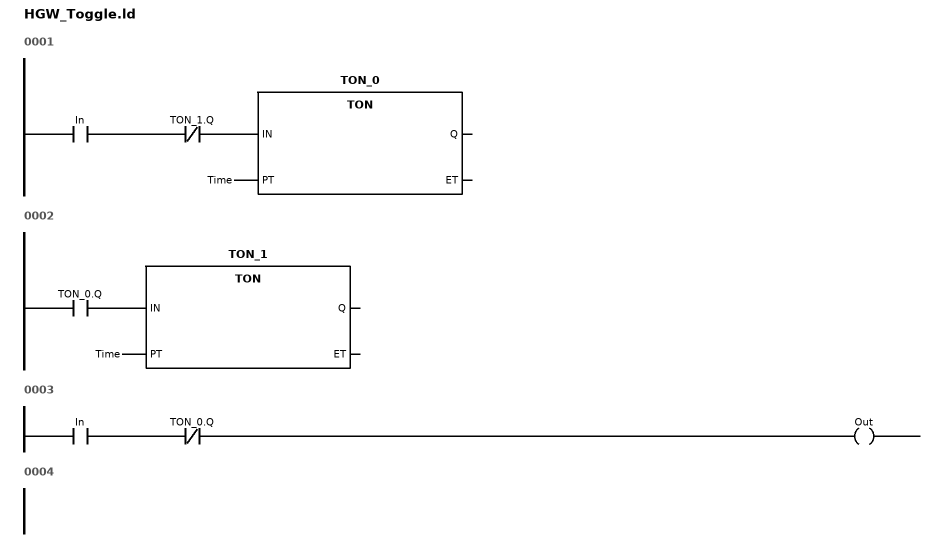
Ladder, written as Structured Text:
```iecst
FUNCTION_BLOCK HGW_Toggle
(* Network 1 *)
TON_0(IN := In AND NOT TON_1.Q, PT := Time);

(* Network 2 *)
TON_1(IN := TON_0.Q, PT := Time);

(* Network 3 *)
Out := In AND NOT TON_0.Q;

(* Network 4 *)
END_FUNCTION_BLOCK
```

### Library Logical/Libraries/CSV_File (IEC, version 2.01.7)
Depends on: AsMath, AsMem, AsString, FileIO, runtime, standard, sys_lib, astime

#### CSV_File.fun
```iecst
FUNCTION_BLOCK CSV_CheckFile
VAR
		statusInternal	:UINT;
		fileVersionStr	:STRING[255];
		cntSizesFound	:USINT;
		ixCmp	:USINT;
		pSize	: REFERENCE TO UDINT;
		SizesFound	:ARRAY [0..254] OF UDINT;
		fileOffset	:UDINT;
		sizeSignificationStr	:STRING[255];
		lineBuf	:STRING[255];
		versionFound	:BOOL;
		maxLenLine	:UINT;
		ixLine	:UDINT;
		ixLineMax	:UDINT;
		lineCnt	:UDINT;
		FClose	:FileClose;
		fileIdent	:UDINT;
		pChar	: REFERENCE TO USINT;
		FOpen	:FileOpen;
		FRead	:FileRead;
		verSignificationStr	:STRING[255];
		R_TRIG_0	:R_TRIG;
		fileCheckStep	:UINT;
		CharPerCyclic	:USINT;
	END_VAR
	VAR_INPUT
		enable	:BOOL;
		pFileName	:UDINT;
		pDevice	:UDINT;
		pStructSizes	:UDINT;
		NumOfStruct	:USINT;
		pVersion	:UDINT;
		pFileBuffer	:UDINT;
		FileBufferSize	:UDINT;
	END_VAR
	VAR_OUTPUT
		status	:UINT;
		fileError	:UINT;
	END_VAR
END_FUNCTION_BLOCK
FUNCTION_BLOCK CSV_InitCheckFile
VAR
		AsMemPartAlloc_0	:AsMemPartAlloc;
		AsMemPartCreate_0	:AsMemPartCreate;
	END_VAR
	VAR_INPUT
		enable	:BOOL;
		MemCounter	:UDINT;
	END_VAR
	VAR_OUTPUT
		status	:UINT;
		pFileBuffer	:UDINT;
		FileBufferSize	:UDINT;
	END_VAR
END_FUNCTION_BLOCK
FUNCTION_BLOCK CSV_Search
VAR
		Internal	:_csv_search_internal;
		zzDTGetTime00000	:DTGetTime;
		SearchChar	: REFERENCE TO USINT;
		Dyn_Bool	: REFERENCE TO BOOL;
		Dyn_Usint	: REFERENCE TO USINT;
		Dyn_Sint	: REFERENCE TO SINT;
		Dyn_Uint	: REFERENCE TO UINT;
		Dyn_Int	: REFERENCE TO INT;
		Dyn_Udint	: REFERENCE TO UDINT;
		Dyn_Dint	: REFERENCE TO DINT;
		Dyn_Real	: REFERENCE TO REAL;
		Dyn_Date_and_Time	: REFERENCE TO DATE_AND_TIME;
		Dyn_Time	: REFERENCE TO TIME;
		OnlyOneVar	:BOOL;
	END_VAR
	VAR_INPUT
		pStructName	:UDINT;
		NumOfStructs	:USINT;
		pStructMem	:UDINT;
		MemLen	:UDINT;
		Options	:UDINT;
		FullNameLenght	:BOOL;
		FileHeader	:BOOL;
		Separator	:USINT;
		pMaschineNo	:UDINT;
		pComment	:UDINT;
		pVersion	:UDINT;
	END_VAR
	VAR_OUTPUT
		status	:UINT;
		ErrorName	:USINT;
		FileLen	:UDINT;
	END_VAR
END_FUNCTION_BLOCK
FUNCTION_BLOCK CSV_Init
VAR
		Internal	:_csv_init_Internal;
		SearchChar	: REFERENCE TO USINT;
		Dyn_Usint	: REFERENCE TO USINT;
		Dyn_Sint	: REFERENCE TO SINT;
		Dyn_Int	: REFERENCE TO INT;
		Dyn_Dint	: REFERENCE TO DINT;
		Dyn_Uint	: REFERENCE TO UINT;
		Dyn_Udint	: REFERENCE TO UDINT;
		Dyn_Real	: REFERENCE TO REAL;
		Dyn_Date_and_Time	: REFERENCE TO DATE_AND_TIME;
		Dyn_Time	: REFERENCE TO TIME;
		OnlyOneVar	:BOOL;
	END_VAR
	VAR_INPUT
		pStructName	:UDINT;
		NumOfStructs	:USINT;
		FullNameLenght	:BOOL;
		Options	:UDINT;
	END_VAR
	VAR_OUTPUT
		status	:UINT;
		ErrorName	:USINT;
		pStructMem	:UDINT;
		MemCounter	:UDINT;
	END_VAR
END_FUNCTION_BLOCK
FUNCTION_BLOCK CSV_ListFile
VAR
		DirRead_01	:DirRead;
		DirInfo_01	:DirInfo;
		TmpString	:ARRAY [0..50] OF USINT;
		Step	:USINT;
		i	:UINT;
		TmpExtension	:STRING[4];
		FileInfo	:fiDIR_READ_DATA;
		result1	:DINT;
		result2	:DINT;
		FileNumAct	:UINT;
		FileNumOnDisk	:UINT;
		Offset	:UDINT;
		pActName	:UDINT;
		dateandtime	:DTStructure;
		UpLines	:UINT;
		DownLines	:UINT;
		PosFirstLine	:UINT;
		OptionStruct	: REFERENCE TO CSV_ListFileOption_typ;
	END_VAR
	VAR_INPUT
		pStringArray	:UDINT;
		SizeStringArray	:UDINT;
		ArrayNum	:UINT;
		NumListboxLines	:UINT;
		pFileDevice	:UDINT;
		pPath	:UDINT;
		MaxNameLenght	:USINT;
		SetFocusPos	:UINT;
		command	:USINT;
	END_VAR
	VAR_OUTPUT
		status	:UINT;
		CSV_FileNum	:UINT;
		ListboxFocusPos	:UINT;
		ScrollUp	:BOOL;
		ScrollDown	:BOOL;
	END_VAR
END_FUNCTION_BLOCK
FUNCTION_BLOCK SearchFileName
VAR
		step	:USINT;
		FileName	:STRING[40];
		i	:USINT;
		FileOpen_01	:FileOpen;
		FileClose_01	:FileClose;
		SearchChar	: REFERENCE TO USINT;
	END_VAR
	VAR_INPUT
		pFileName	:UDINT;
		pDevice	:UDINT;
	END_VAR
	VAR_OUTPUT
		status	:UINT;
	END_VAR
END_FUNCTION_BLOCK
FUNCTION_BLOCK CSV_ReadFile
VAR
		FileOpen_CSV	:FileOpen;
		FileRead_CSV	:FileRead;
		FileClose_CSV	:FileClose;
		Internal	:_csv_read_internal;
		Dyn_Usint	: REFERENCE TO USINT;
		SearchChar	: REFERENCE TO USINT;
		Dyn_Bool	: REFERENCE TO BOOL;
		Dyn_Sint	: REFERENCE TO SINT;
		Dyn_Uint	: REFERENCE TO UINT;
		Dyn_Int	: REFERENCE TO INT;
		Dyn_Udint	: REFERENCE TO UDINT;
		Dyn_Dint	: REFERENCE TO DINT;
		Dyn_String	: REFERENCE TO STRING[80];
		Dyn_Real	: REFERENCE TO REAL;
		Dyn_Date_and_Time	: REFERENCE TO DATE_AND_TIME;
		Dyn_Time	: REFERENCE TO TIME;
		Part	:BOOL;
		TestUsint	:USINT;
		temp_status	:UINT;
	END_VAR
	VAR_INPUT
		pFileName	:UDINT;
		pDevice	:UDINT;
		pPath	:UDINT;
		No_DatatypControl	:BOOL;
		Separator	:USINT;
		IgnoreError	:BOOL;
		Options	:UDINT;
	END_VAR
	VAR_OUTPUT
		status	:UINT;
		LineCnt	:UDINT;
		VarCnt	:UDINT;
		ErrorLine	:UDINT;
		ErrorNumber	:UINT;
		ErrorCnt	:UDINT;
	END_VAR
END_FUNCTION_BLOCK
FUNCTION_BLOCK ExListFile
VAR
		Internal	:_csv_exfilelist_internal;
		DirInfo_CSV	:DirInfo;
		DirRead_CSV	:DirRead;
		FileOpen_CSV	:FileOpen;
		FileRead_CSV	:FileRead;
		FileClose_CSV	:FileClose;
		DynUsint	: REFERENCE TO USINT;
	END_VAR
	VAR_INPUT
		pStringArray	:UDINT;
		SizeStringArray	:UDINT;
		NumListboxLines	:UINT;
		ArrayNum	:UINT;
		pFileDevice	:UDINT;
		MaxNameLenght	:USINT;
		SetFocusPos	:UINT;
		command	:USINT;
		pOptions	:UDINT;
	END_VAR
	VAR_OUTPUT
		status	:UINT;
		CSV_FileNum	:UINT;
		ListboxFocusPos	:UINT;
		ScrollUp	:BOOL;
		ScrollDown	:BOOL;
	END_VAR
END_FUNCTION_BLOCK
FUNCTION_BLOCK CSV_WriteFile
VAR
		Step	:USINT;
		FileCreate_CSV	:FileCreate;
		FileWrite_CSV	:FileWrite;
		FileDelete_CSV	:FileDelete;
		FileClose_CSV	:FileClose;
		FileName	:STRING[80];
		i	:USINT;
		Dyn_Usint	: REFERENCE TO USINT;
		DevMemInfo_CSV	:DevMemInfo;
		Path	:STRING[100];
	END_VAR
	VAR_INPUT
		pFileName	:UDINT;
		pDevice	:UDINT;
		pPath	:UDINT;
		pStructMem	:UDINT;
		MemLen	:UDINT;
		Mode	:USINT;
	END_VAR
	VAR_OUTPUT
		status	:UINT;
	END_VAR
END_FUNCTION_BLOCK
```

### Package Logical/HMI - HMI Related Code

### Program Logical/HMI/Splash (IEC) - HMI Splash Screen Control

#### SplashCyclic.st
```iecst
(********************************************************************
 * COPYRIGHT --
 ********************************************************************
 * Program: Splash
 * File: SplashCyclic.st
 * Author: pkiel
 * Created: October 09, 2009
 ********************************************************************
 * Implementation of program Splash
 ********************************************************************)

PROGRAM _CYCLIC

(* MAIN SCREEEN *)
	(* Get Handle For Main HMI *)
		IF Ready <> 1 THEN
		 	VC_HANDLE:= VA_Setup(1,'HMI_10');
		 	IF (VC_HANDLE <> 0) THEN
		 		Ready:= 1;
			END_IF
		END_IF

	(* Monitor To See If Main HMI Screen Calibration Is Active *)
		 IF (Ready = 1) THEN
		 	IF (VA_Saccess(1,VC_HANDLE)= 0) THEN
			 	Status:= VA_GetCalStatus (1,VC_HANDLE);
		 		VA_Srelease(1,VC_HANDLE);
			END_IF
		END_IF

	(* Main HMI Splash Screen Control *)
		IF (gCurrentScreen=0 AND Status=0) THEN
			TON_0( IN:=NOT SplashDone, PT:=T#12s );
			ElapsedTime:=TIME_TO_REAL(TON_0.ET);
			CountDown:=12-(ElapsedTime/1000);
			SplashDone:=TON_0.Q;
			IF (TON_0.Q) THEN
				gScreenControl:=1;
        g_bSplashDone := 1 ;
			END_IF
		END_IF

END_PROGRAM
```

### Program Logical/HMI/HMI_Control (IEC) - General HMI Control

#### HMI_ControlCyclic.st - Cyclic code
```iecst
(********************************************************************
 * COPYRIGHT --
 ********************************************************************
 * Program: HMI_Control
 * File: HMI_ControlCyclic.st
 * Author: pkiel
 * Created: September 17, 2009
 ********************************************************************
 * Implementation of program HMI_Control
 ********************************************************************)

PROGRAM _CYCLIC

(* Screen GoTo Control on Main HMI For Main, Setup, & Status Screens *)
	IF (gHMI_GoToMain_PB) THEN
		gScreenControl:=HMI_MainScreenGroup;
		gHMI_GoToMain_PB:=0;
		HMI_ScreenGroup_Ind:=0;
		gHMI_PasswordLevel:=0;
	END_IF;
	IF (gHMI_GoToSetup_PB) THEN
		gScreenControl:=HMI_SetupScreenGroup;
		gHMI_GoToSetup_PB:=0;
		HMI_ScreenGroup_Ind:=1;
		gHMI_PasswordLevel:=0;
	END_IF;
	IF (gHMI_GoToStatus_PB) THEN
		gScreenControl:=20;
		gHMI_GoToStatus_PB:=0;
		HMI_ScreenGroup_Ind:=2;
		gHMI_PasswordLevel:=0;
	END_IF;
	IF (gHMI_GoToAlarm_PB) THEN
		gScreenControl:=30;
		gHMI_GoToAlarm_PB:=0;
		HMI_ScreenGroup_Ind:=4;
		gHMI_PasswordLevel:=0;
	END_IF;
  IF (gHMI_GoToMaint_PB) THEN
    gScreenControl:=HMI_MaintenanceScreenGroup;
    gMaintDropdown := gScreenControl;
    gHMI_GoToMaint_PB:=0;
    HMI_ScreenGroup_Ind:=3;
  END_IF;
  IF (gHMI_GoToHoldTearDrum_PB) THEN
    gScreenControl:=12;
    gHMI_GoToHoldTearDrum_PB:=0;
  END_IF;
	CASE (HMI_ScreenGroup_Ind) OF
		0:
			HMI_MainScreenGroup:=gCurrentScreen;
			HMI_MainScreenGroup:=LIMIT(1,HMI_MainScreenGroup,6);
		1:
			HMI_SetupScreenGroup:=gCurrentScreen;
			HMI_SetupScreenGroup:=LIMIT(10,HMI_SetupScreenGroup,12);

		2:
			HMI_StatusScreenGroup:=gCurrentScreen;
			HMI_StatusScreenGroup:=LIMIT(20,HMI_StatusScreenGroup,20);
		3:
			IF (gMaintScreenChange) THEN
				gScreenControl := gMaintDropdown;
				gMaintScreenChange :=0;
			END_IF
			HMI_MaintenanceScreenGroup:=gCurrentScreen;
			HMI_MaintenanceScreenGroup:=LIMIT(40,HMI_MaintenanceScreenGroup,57);
	END_CASE;

(* Transfers for Servo Status Screens *)
	HMI_Status_Ind:=LIMIT(0,HMI_Status_Ind,15);
	IF (gCurrentScreen=20) THEN
			gA[HMI_Status_Ind].ErrorAck			:=	HMI_ErrorAck;
			HMI_ErrorCount				:=	gA[HMI_Status_Ind].ErrorCount;
			HMI_ErrorText				:=	gA[HMI_Status_Ind].ErrorText;
			HMI_Ind_Enabled				:=	gA[HMI_Status_Ind].Ind_Enabled;
			HMI_Ind_InMotion			:=	gA[HMI_Status_Ind].Ind_InMotion;
			HMI_Error					:=	gA[HMI_Status_Ind].Error;
			HMI_ErrorStop				:=	gA[HMI_Status_Ind].ErrorStop;
			HMI_ErrorID					:=	gA[HMI_Status_Ind].ErrorID;
			HMI_Ind_DiscreteMotion		:=	gA[HMI_Status_Ind].Ind_DiscreteMotion;
			HMI_Ind_ContinuousMotion	:=	gA[HMI_Status_Ind].Ind_ContinuousMotion;
			HMI_Ind_SynchronizedMotion	:=	gA[HMI_Status_Ind].Ind_SynchronizedMotion;
			HMI_Ind_NetworkInit			:=	gA[HMI_Status_Ind].Ind_NetworkInit;
			HMI_Ind_ControllerStatus	:=	gA[HMI_Status_Ind].Ind_ControllerStatus;
			HMI_Ind_Homed				:=	gA[HMI_Status_Ind].Ind_Homed;
			HMI_Input_Home				:=	gA[HMI_Status_Ind].Input_Home;
			HMI_Input_DriveEnable		:=	gA[HMI_Status_Ind].Input_DriveEnable;
			HMI_Input_Trigger1			:=	gA[HMI_Status_Ind].Input_Trigger1;
			HMI_Input_Trigger2			:=	gA[HMI_Status_Ind].Input_Trigger2;
			HMI_PositionInch			:=	gA[HMI_Status_Ind].PositionInch;
			HMI_PositionDeg				:=	gA[HMI_Status_Ind].PositionDeg;
			HMI_ActualVelocity			:=	gA[HMI_Status_Ind].ActualVelocity;
	END_IF

(*Data Entry Lockout*)
	IF (gA[9].Ind_InMotion) THEN
		DataLock_Motion := 2;
  ELSE
    DataLock_Motion := 0;
	END_IF

// Display curve max speed Perf
  IF HMI_bMaxSpeedPerf_PB THEN
    HMI_iSelCurvMaxSpeedPerf := gInchMetric_Ind ;
    HMI_uiCurvVisibl := 0 ; // Curve visible
  ELSE
    HMI_iSelCurvMaxSpeedPerf := 0 ;
    HMI_uiCurvVisibl := 1 ; // Curve unvisible
  END_IF
  IF (gCurrentScreen <> 11) THEN
    HMI_bMaxSpeedPerf_PB := 0 ;
  END_IF

// Hide Holding Tearing Envelope Bag Offset
  IF (gCurrentScreen <> 1) THEN
    HMI_iHTEnvBOffsetVisibl := 1 ;
  END_IF

// ----------------------------------------------------------------------------------------
// Picture animation

    // Sychro axis animation
    IF g_bSynchroAxisInProgress THEN
      iCountCycl := iCountCycl + 1 ;
      IF (iCountCycl >= 3) THEN      // HMI_Control Task time = 0,1s. Animation => 25 pictures/s => Cycle count >= 2.5 (=>3)
        iCountCycl := 0 ;
        iAnimStep  := iAnimStep + 1 ;
        HMI_iAnimSynchroAxis := iAnimStep ;
        IF (iAnimStep >= 4) THEN
          iAnimStep := 0 ;
        END_IF
      END_IF
      HMI_iAnimSynchroAxisVisibl := 0 ;    // Visible
    ELSE
      iCountCycl := 0 ;
      iAnimStep  := 0 ;
      HMI_iAnimSynchroAxis := 0 ;
      HMI_iAnimSynchroAxisVisibl := 1 ;    // Not visible
    END_IF

    // Help view axis config
    IF NOT(HMI_bPBShowEnvBConf) THEN
      IF HMI_iAnimPictHoldTearEnvB > 2 THEN
        HMI_iAnimPictHoldTearEnvB := 1 ;
      END_IF
      IF HMI_iAnimPictHoldTearEnvB < 1 THEN
        HMI_iAnimPictHoldTearEnvB := 2 ;
      END_IF
      HMI_iAnimTubLVisibl := 0 ; // Visible

      CASE HMI_iAnimPictHoldTearEnvB OF
        1 :
          HMI_iAnimHoldTearEnvB_1 := 1 ;
          HMI_iAnimHoldTearEnvB_2 := 2 ;
          HMI_rTubLInf_1 := g_rMinBagSize_RS26_mm/25.4 ;
          HMI_rTubLSup_1 := gr_rBagSize4_2Pliers_mm/25.4 ;
          HMI_rTubLInf_2 := gr_rBagSize4_2Pliers_mm/25.4 ;
          HMI_rTubLSup_2 := gr_rEnvBSizeTear2_1_mm/25.4 ;
          HMI_iNumbPliers_1 := 4 ;
          HMI_iNumbPliers_2 := 2 ;
          HMI_iAnimPict2Visibl := 0 ;
        2 :
          HMI_iAnimHoldTearEnvB_1 := 3 ;
          HMI_iAnimHoldTearEnvB_2 := 0 ;
          HMI_rTubLInf_1 := gr_rEnvBSizeTear2_1_mm/25.4 ;
          HMI_rTubLSup_1 := g_rMaxBagSize_RS26_mm/25.4 ;
          HMI_rTubLInf_2 := 0.0 ;
          HMI_rTubLSup_2 := 0.0 ;
          HMI_iNumbPliers_1 := 2 ;
          HMI_iNumbPliers_2 := 0 ;
          HMI_iAnimPict2Visibl := 1 ; // Hide
      END_CASE
      rPosHoldEnvB := gr_rPosEnvBHoldBag + 45.0 ;
      HMI_rPosHoldEnvB := H_FC_Modulus (
                               IN_rMod := 360.0 ,
                               IN_rVar := rPosHoldEnvB
                                       ) ;
    ELSE
      HMI_iAnimTubLVisibl     := 1 ; // Hide
      HMI_iAnimHoldTearEnvB_1 := 4 ;
      HMI_iAnimHoldTearEnvB_2 := 5 ;
      HMI_rTubLInf_1 := g_rMinBagSize_EnvB_mm/25.4 ;
      HMI_rTubLSup_1 := gr_rBagSize1_2Hold_mm/25.4 ;
      HMI_rTubLInf_2 := gr_rBagSize1_2Hold_mm/25.4 ;
      HMI_rTubLSup_2 := g_rMaxBagSize_EnvB_mm/25.4 ;
      HMI_iNumbPliers_1 := 2 ;
      HMI_iNumbPliers_2 := 2 ;
      HMI_iAnimPict2Visibl := 0 ;
      HMI_rPosHoldEnvB := gr_rPosEnvBHoldBag ;
    END_IF

END_PROGRAM
```

#### HMI_ControlInit.st - Initialization code
```iecst
(********************************************************************
 * COPYRIGHT --
 ********************************************************************
 * Program: HMI_Control
 * File: HMI_ControlInit.st
 * Author: pkiel
 * Created: September 17, 2009
 ********************************************************************
 * Implementation of program HMI_Control
 ********************************************************************)

PROGRAM _INIT

	HMI_MainScreenGroup:=1;
	HMI_SetupScreenGroup:=10;
	HMI_StatusScreenGroup:=20;
	HMI_MaintenanceScreenGroup:=40;
	HMI_AlarmInputStatus:=HMI_AlarmInputStatus;
  HMI_uiCurvVisibl := 1 ;
  HMI_uiNeverVisibl := 1 ;

  // Unwinder
  HMI_strMP_UNW_HydroPump    := '21Q1' ;
  // Flexo Press
  HMI_strMP_FP_MotorFan      := '73Q2' ;
  HMI_strMP_FP_SlowRot1      := '27Q1' ;
  HMI_strMP_FP_SlowRot2      := '27Q2' ;
  HMI_strMP_FP_SlowRot3      := '27Q3' ;
  HMI_strMP_FP_SlowRot4      := '27Q4' ;
  HMI_strMP_FP_SlowRot5      := '28Q1' ;
  HMI_strMP_FP_SlowRot6      := '28Q2' ;
  // Bag Machine
  HMI_strMP_GlueSlowRotation := '19Q1' ;
  HMI_strMP_PerfFan          := '73Q4' ;
  HMI_strMP_Vacuum           := '14Q1' ;
  // 3-Web unit
  HMI_strMP_3W_MotorFan      := '36Q1' ;
  // Dryer
  HMI_strMP_DRY_Blower       := '31Q1 OR 31Q2' ;
  HMI_strMP_DRY_Heater       := '3Q5' ;
  HMI_strSS_DRY_Thermostat   := '79F1' ;
  // Cold Micro Perf Waste suction
  HMI_strMP_CMP_WasteSuc     := '15Q2' ;
  // Envelope Bag Waste Suction
  HMI_strMP_EB_WasteSuc      := '36Q1' ;

  HMI_iAnimSynchroAxisVisibl := 1 ;
  g_bSplashDone := 0 ;

  HMI_iHTEnvBOffsetVisibl := 1 ;

	// Initialize Default Gateway...RS26 Pyrollpack_14661 IP Config IP Adresse  : 10.0.1.67
  //                                                               Gateway    : 10.0.1.1
  //                                                               SubNetMask : 255.255.255.0
	CfgSetDefaultGateway_0(enable := 1 , pDevice := ADR('IF5'), pGateway := ADR('10.0.1.1'), Option := 1);

END_PROGRAM
```

#### HMI_Control.var - Local variables
```iecst
(********************************************************************
 * COPYRIGHT --
 ********************************************************************
 * Program: HMI_Control
 * File: HMI_Control.var
 * Author: pkiel
 * Created: September 17, 2009
 ********************************************************************
 * Local variables of program HMI_Control
 ********************************************************************)
VAR
	CfgSetDefaultGateway_0 : CfgSetDefaultGateway;
	DataLock_Motion : UINT;
	HMI_ActualVelocity : REAL;
	HMI_AlarmFilterControl : INT;
	HMI_AlarmFilterGroup : INT;
	HMI_AlarmInputStatus : INT;
	HMI_Error : BOOL;
	HMI_ErrorAck : BOOL;
	HMI_ErrorCount : UINT;
	HMI_ErrorID : UINT;
	HMI_ErrorStop : BOOL;
	HMI_ErrorText : ARRAY[0..3] OF STRING[79];
	HMI_Ind_ContinuousMotion : BOOL;
	HMI_Ind_ControllerStatus : BOOL;
	HMI_Ind_DiscreteMotion : BOOL;
	HMI_Ind_Enabled : BOOL;
	HMI_Ind_Homed : BOOL;
	HMI_Ind_InMotion : BOOL;
	HMI_Ind_NetworkInit : BOOL;
	HMI_Ind_SynchronizedMotion : BOOL;
	HMI_Input_DriveEnable : BOOL;
	HMI_Input_Home : BOOL;
	HMI_Input_Trigger1 : BOOL;
	HMI_Input_Trigger2 : BOOL;
	HMI_MainScreenGroup : UINT;
	HMI_MaintenanceScreenGroup : UINT;
	HMI_PositionDeg : REAL;
	HMI_PositionInch : REAL;
	HMI_Screen2Group_Ind : UINT;
	HMI_ScreenGroup_Ind : UINT;
	HMI_SetupScreenGroup : UINT;
	HMI_Status_Ind : UINT;
  HMI_StatusScreenGroup : UINT;
  HMI_bMaxSpeedPerf_PB : BOOL;
  HMI_iSelCurvMaxSpeedPerf : INT;
  HMI_uiCurvVisibl         : UINT;
  HMI_uiNeverVisibl        : UINT := 1 ;

  HMI_strMP_UNW_HydroPump    : STRING[10] ;
  HMI_strMP_FP_MotorFan      : STRING[10] ;
  HMI_strMP_FP_SlowRot1      : STRING[10] ;
  HMI_strMP_FP_SlowRot2      : STRING[10] ;
  HMI_strMP_FP_SlowRot3      : STRING[10] ;
  HMI_strMP_FP_SlowRot4      : STRING[10] ;
  HMI_strMP_FP_SlowRot5      : STRING[10] ;
  HMI_strMP_FP_SlowRot6      : STRING[10] ;
  HMI_strMP_GlueSlowRotation : STRING[10] ;
  HMI_strMP_PerfFan          : STRING[10] ;
  HMI_strMP_Vacuum           : STRING[10] ;
  HMI_strMP_3W_MotorFan      : STRING[10] ;
  HMI_strMP_DRY_Blower       : STRING[12] ;
  HMI_strMP_DRY_Heater       : STRING[10] ;
  HMI_strSS_DRY_Thermostat   : STRING[10] ;
  HMI_strMP_CMP_WasteSuc     : STRING[10] ;
  HMI_strMP_EB_WasteSuc      : STRING[10] ; (*Envelope Bag Waste Suction*)

  HMI_iAnimHoldTearEnvB_1 : INT ;
  HMI_iAnimHoldTearEnvB_2 : INT ;
  HMI_iNumbPliers_1 : INT ;
  HMI_iNumbPliers_2 : INT ;
  HMI_iAnimPictHoldTearEnvB : INT ;
  HMI_bPBShowEnvBConf : BOOL ;
  HMI_rTubLInf_1 : REAL ;
  HMI_rTubLInf_2 : REAL ;
  HMI_rTubLSup_1 : REAL ;
  HMI_rTubLSup_2 : REAL ;
  HMI_iAnimPict2Visibl : INT ;
  HMI_iAnimTubLVisibl : INT ;
  HMI_rPosHoldEnvB : REAL ;
  rPosHoldEnvB : REAL ;

  HMI_iAnimSynchroAxis       :  INT ;
  HMI_iAnimSynchroAxisVisibl : INT ;

  HMI_iHTEnvBOffsetVisibl : INT ;

  iAnimStep   : INT ;
  iCountCycl  : INT ;
  iIndex      : INT ;
END_VAR
```

### Program Logical/HMI/Units (IEC) - HMI Inch/Metric Control
